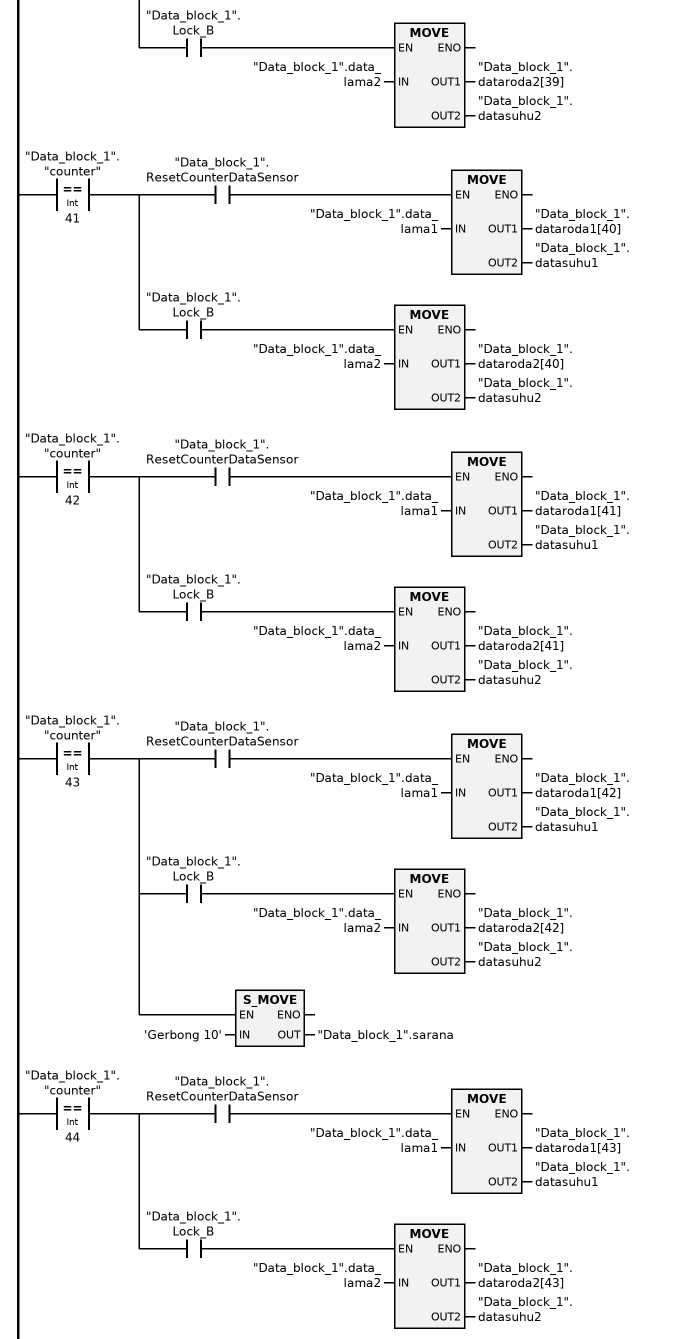
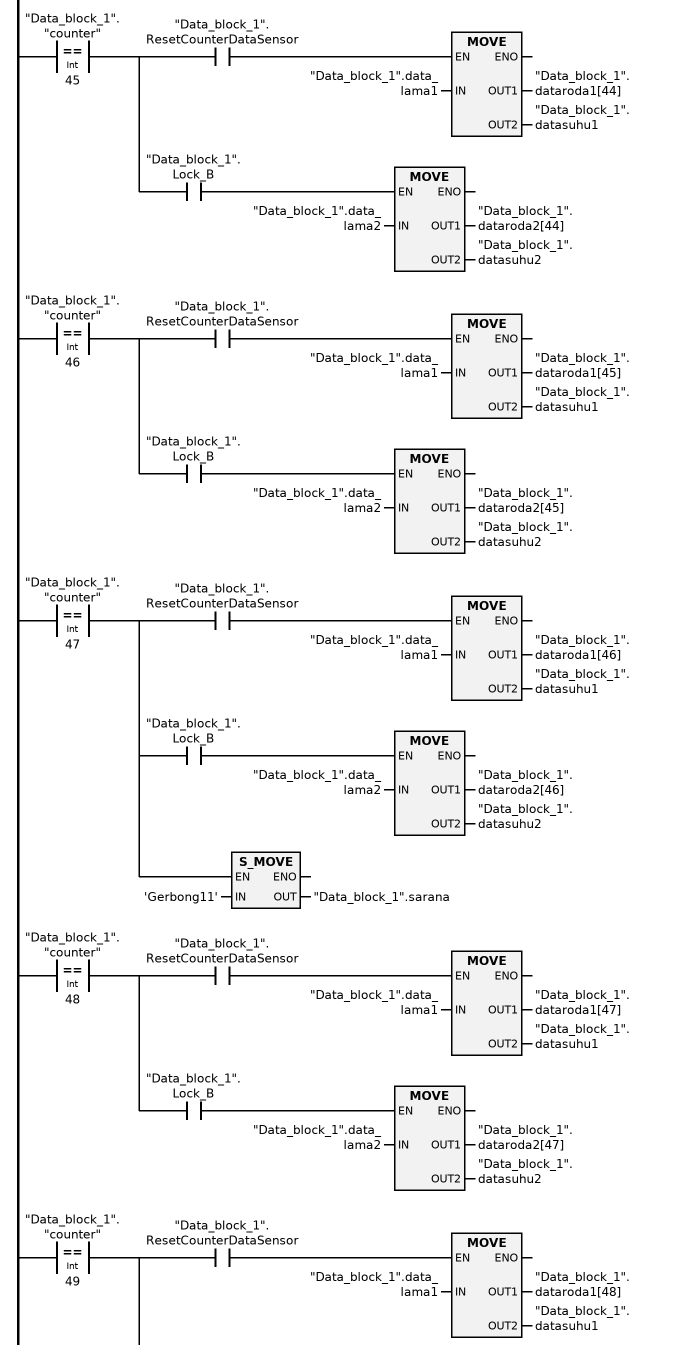
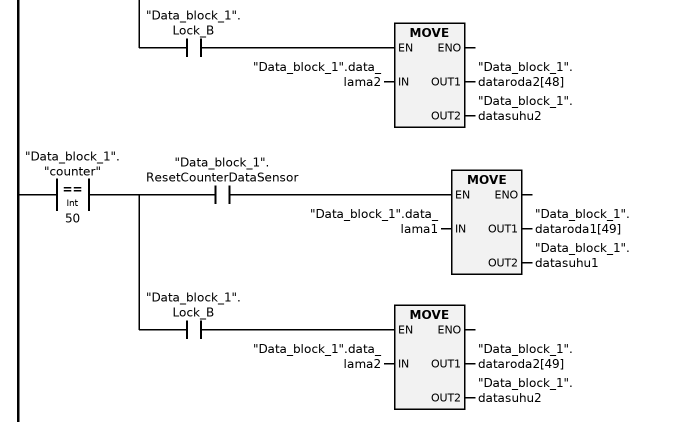
   #_w1 := "Data_block_1"."counter" = 1;
   IF #_w1 AND "Data_block_1".ResetCounterDataSensor THEN
       "Data_block_1".dataroda1[0] := "Data_block_1".data_lama1;
       "Data_block_1".datasuhu1 := "Data_block_1".data_lama1;
   END_IF;
   IF #_w1 AND "Data_block_1".Lock_B THEN
       "Data_block_1".dataroda2[0] := "Data_block_1".data_lama2;
       "Data_block_1".datasuhu2 := "Data_block_1".data_lama2;
   END_IF;
   IF #_w1 THEN S_MOVE(in := 'Lokomotif', out => "Data_block_1".sarana); END_IF;
   #_w2 := "Data_block_1"."counter" = 2;
   IF #_w2 AND "Data_block_1".ResetCounterDataSensor THEN
       "Data_block_1".dataroda1[1] := "Data_block_1".data_lama1;
       "Data_block_1".datasuhu1 := "Data_block_1".data_lama1;
   END_IF;
   IF #_w2 AND "Data_block_1".Lock_B THEN
       "Data_block_1".dataroda2[1] := "Data_block_1".data_lama2;
       "Data_block_1".datasuhu2 := "Data_block_1".data_lama2;
   END_IF;
   #_w3 := "Data_block_1"."counter" = 3;
   IF #_w3 AND "Data_block_1".ResetCounterDataSensor THEN
       "Data_block_1".dataroda1[2] := "Data_block_1".data_lama1;
       "Data_block_1".datasuhu1 := "Data_block_1".data_lama1;
   END_IF;
   IF #_w3 AND "Data_block_1".Lock_B THEN
       "Data_block_1".dataroda2[2] := "Data_block_1".data_lama2;
       "Data_block_1".datasuhu2 := "Data_block_1".data_lama2;
   END_IF;
   #_w4 := "Data_block_1"."counter" = 4;
   IF #_w4 AND "Data_block_1".ResetCounterDataSensor THEN
       "Data_block_1".dataroda1[3] := "Data_block_1".data_lama1;
       "Data_block_1".datasuhu1 := "Data_block_1".data_lama1;
   END_IF;
   IF #_w4 AND "Data_block_1".Lock_B THEN
       "Data_block_1".dataroda2[3] := "Data_block_1".data_lama2;
       "Data_block_1".datasuhu2 := "Data_block_1".data_lama2;
   END_IF;
   #_w5 := "Data_block_1"."counter" = 5;
   IF #_w5 AND "Data_block_1".ResetCounterDataSensor THEN
       "Data_block_1".dataroda1[4] := "Data_block_1".data_lama1;
       "Data_block_1".datasuhu1 := "Data_block_1".data_lama1;
   END_IF;
   IF #_w5 AND "Data_block_1".Lock_B THEN
       "Data_block_1".dataroda2[4] := "Data_block_1".data_lama2;
       "Data_block_1".datasuhu2 := "Data_block_1".data_lama2;
   END_IF;
   #_w6 := "Data_block_1"."counter" = 6;
   IF #_w6 AND "Data_block_1".ResetCounterDataSensor THEN
       "Data_block_1".dataroda1[5] := "Data_block_1".data_lama1;
       "Data_block_1".datasuhu1 := "Data_block_1".data_lama1;
   END_IF;
   IF #_w6 AND "Data_block_1".Lock_B THEN
       "Data_block_1".dataroda2[5] := "Data_block_1".data_lama2;
       "Data_block_1".datasuhu2 := "Data_block_1".data_lama2;
   END_IF;
   #_w7 := "Data_block_1"."counter" = 7;
   IF #_w7 AND "Data_block_1".ResetCounterDataSensor THEN
       "Data_block_1".dataroda1[6] := "Data_block_1".data_lama1;
       "Data_block_1".datasuhu1 := "Data_block_1".data_lama1;
   END_IF;
   IF #_w7 AND "Data_block_1".Lock_B THEN
       "Data_block_1".dataroda2[6] := "Data_block_1".data_lama2;
       "Data_block_1".datasuhu2 := "Data_block_1".data_lama2;
   END_IF;
   IF #_w7 THEN S_MOVE(in := 'Gerbong 1', out => "Data_block_1".sarana); END_IF;
   #_w8 := "Data_block_1"."counter" = 8;
   IF #_w8 AND "Data_block_1".ResetCounterDataSensor THEN
       "Data_block_1".dataroda1[7] := "Data_block_1".data_lama1;
       "Data_block_1".datasuhu1 := "Data_block_1".data_lama1;
   END_IF;
   IF #_w8 AND "Data_block_1".Lock_B THEN
       "Data_block_1".dataroda2[7] := "Data_block_1".data_lama2;
       "Data_block_1".datasuhu2 := "Data_block_1".data_lama2;
   END_IF;
   #_w9 := "Data_block_1"."counter" = 9;
   IF #_w9 AND "Data_block_1".ResetCounterDataSensor THEN
       "Data_block_1".dataroda1[8] := "Data_block_1".data_lama1;
       "Data_block_1".datasuhu1 := "Data_block_1".data_lama1;
   END_IF;
   IF #_w9 AND "Data_block_1".Lock_B THEN
       "Data_block_1".dataroda2[8] := "Data_block_1".data_lama2;
       "Data_block_1".datasuhu2 := "Data_block_1".data_lama2;
   END_IF;
   #_w10 := "Data_block_1"."counter" = 10;
   IF #_w10 AND "Data_block_1".ResetCounterDataSensor THEN
       "Data_block_1".dataroda1[9] := "Data_block_1".data_lama1;
       "Data_block_1".datasuhu1 := "Data_block_1".data_lama1;
   END_IF;
   IF #_w10 AND "Data_block_1".Lock_B THEN
       "Data_block_1".dataroda2[9] := "Data_block_1".data_lama2;
       "Data_block_1".datasuhu2 := "Data_block_1".data_lama2;
   END_IF;
   #_w11 := "Data_block_1"."counter" = 11;
   IF #_w11 AND "Data_block_1".ResetCounterDataSensor THEN
       "Data_block_1".dataroda1[10] := "Data_block_1".data_lama1;
       "Data_block_1".datasuhu1 := "Data_block_1".data_lama1;
   END_IF;
   IF #_w11 AND "Data_block_1".Lock_B THEN
       "Data_block_1".dataroda2[10] := "Data_block_1".data_lama2;
       "Data_block_1".datasuhu2 := "Data_block_1".data_lama2;
   END_IF;
   IF #_w11 THEN S_MOVE(in := 'Gerbong 2', out => "Data_block_1".sarana); END_IF;
   #_w12 := "Data_block_1"."counter" = 12;
   IF #_w12 AND "Data_block_1".ResetCounterDataSensor THEN
       "Data_block_1".dataroda1[11] := "Data_block_1".data_lama1;
       "Data_block_1".datasuhu1 := "Data_block_1".data_lama1;
   END_IF;
   IF #_w12 AND "Data_block_1".Lock_B THEN
       "Data_block_1".dataroda2[11] := "Data_block_1".data_lama2;
       "Data_block_1".datasuhu2 := "Data_block_1".data_lama2;
   END_IF;
   #_w13 := "Data_block_1"."counter" = 13;
   IF #_w13 AND "Data_block_1".ResetCounterDataSensor THEN
       "Data_block_1".dataroda1[12] := "Data_block_1".data_lama1;
       "Data_block_1".datasuhu1 := "Data_block_1".data_lama1;
   END_IF;
   IF #_w13 AND "Data_block_1".Lock_B THEN
       "Data_block_1".dataroda2[12] := "Data_block_1".data_lama2;
       "Data_block_1".datasuhu2 := "Data_block_1".data_lama2;
   END_IF;
   #_w14 := "Data_block_1"."counter" = 14;
   IF #_w14 AND "Data_block_1".ResetCounterDataSensor THEN
       "Data_block_1".dataroda1[13] := "Data_block_1".data_lama1;
       "Data_block_1".datasuhu1 := "Data_block_1".data_lama1;
   END_IF;
   IF #_w14 AND "Data_block_1".Lock_B THEN
       "Data_block_1".dataroda2[13] := "Data_block_1".data_lama2;
       "Data_block_1".datasuhu2 := "Data_block_1".data_lama2;
   END_IF;
   #_w15 := "Data_block_1"."counter" = 15;
   IF #_w15 AND "Data_block_1".ResetCounterDataSensor THEN
       "Data_block_1".dataroda1[14] := "Data_block_1".data_lama1;
       "Data_block_1".datasuhu1 := "Data_block_1".data_lama1;
   END_IF;
   IF #_w15 AND "Data_block_1".Lock_B THEN
       "Data_block_1".dataroda2[14] := "Data_block_1".data_lama2;
       "Data_block_1".datasuhu2 := "Data_block_1".data_lama2;
   END_IF;
   IF #_w15 THEN S_MOVE(in := 'Gerbong 3', out => "Data_block_1".sarana); END_IF;
   #_w16 := "Data_block_1"."counter" = 16;
   IF #_w16 AND "Data_block_1".ResetCounterDataSensor THEN
       "Data_block_1".dataroda1[15] := "Data_block_1".data_lama1;
       "Data_block_1".datasuhu1 := "Data_block_1".data_lama1;
   END_IF;
   IF #_w16 AND "Data_block_1".Lock_B THEN
       "Data_block_1".dataroda2[15] := "Data_block_1".data_lama2;
       "Data_block_1".datasuhu2 := "Data_block_1".data_lama2;
   END_IF;
   #_w17 := "Data_block_1"."counter" = 17;
   IF #_w17 AND "Data_block_1".ResetCounterDataSensor THEN
       "Data_block_1".dataroda1[16] := "Data_block_1".data_lama1;
       "Data_block_1".datasuhu1 := "Data_block_1".data_lama1;
   END_IF;
   IF #_w17 AND "Data_block_1".Lock_B THEN
       "Data_block_1".dataroda2[16] := "Data_block_1".data_lama2;
       "Data_block_1".datasuhu2 := "Data_block_1".data_lama2;
   END_IF;
   #_w18 := "Data_block_1"."counter" = 18;
   IF #_w18 AND "Data_block_1".ResetCounterDataSensor THEN
       "Data_block_1".dataroda1[17] := "Data_block_1".data_lama1;
       "Data_block_1".datasuhu1 := "Data_block_1".data_lama1;
   END_IF;
   IF #_w18 AND "Data_block_1".Lock_B THEN
       "Data_block_1".dataroda2[17] := "Data_block_1".data_lama2;
       "Data_block_1".datasuhu2 := "Data_block_1".data_lama2;
   END_IF;
   #_w19 := "Data_block_1"."counter" = 19;
   IF #_w19 AND "Data_block_1".ResetCounterDataSensor THEN
       "Data_block_1".dataroda1[18] := "Data_block_1".data_lama1;
       "Data_block_1".datasuhu1 := "Data_block_1".data_lama1;
   END_IF;
   IF #_w19 AND "Data_block_1".Lock_B THEN
       "Data_block_1".dataroda2[18] := "Data_block_1".data_lama2;
       "Data_block_1".datasuhu2 := "Data_block_1".data_lama2;
   END_IF;
   IF #_w19 THEN S_MOVE(in := 'Gerbong 4', out => "Data_block_1".sarana); END_IF;
   #_w20 := "Data_block_1"."counter" = 20;
   IF #_w20 AND "Data_block_1".ResetCounterDataSensor THEN
       "Data_block_1".dataroda1[19] := "Data_block_1".data_lama1;
       "Data_block_1".datasuhu1 := "Data_block_1".data_lama1;
   END_IF;
   IF #_w20 AND "Data_block_1".Lock_B THEN
       "Data_block_1".dataroda2[19] := "Data_block_1".data_lama2;
       "Data_block_1".datasuhu2 := "Data_block_1".data_lama2;
   END_IF;
   #_w21 := "Data_block_1"."counter" = 21;
   IF #_w21 AND "Data_block_1".ResetCounterDataSensor THEN
       "Data_block_1".dataroda1[20] := "Data_block_1".data_lama1;
       "Data_block_1".datasuhu1 := "Data_block_1".data_lama1;
   END_IF;
   IF #_w21 AND "Data_block_1".Lock_B THEN
       "Data_block_1".dataroda2[20] := "Data_block_1".data_lama2;
       "Data_block_1".datasuhu2 := "Data_block_1".data_lama2;
   END_IF;
   #_w22 := "Data_block_1"."counter" = 22;
   IF #_w22 AND "Data_block_1".ResetCounterDataSensor THEN
       "Data_block_1".dataroda1[21] := "Data_block_1".data_lama1;
       "Data_block_1".datasuhu1 := "Data_block_1".data_lama1;
   END_IF;
   IF #_w22 AND "Data_block_1".Lock_B THEN
       "Data_block_1".dataroda2[21] := "Data_block_1".data_lama2;
       "Data_block_1".datasuhu2 := "Data_block_1".data_lama2;
   END_IF;
   #_w23 := "Data_block_1"."counter" = 23;
   IF #_w23 AND "Data_block_1".ResetCounterDataSensor THEN
       "Data_block_1".dataroda1[22] := "Data_block_1".data_lama1;
       "Data_block_1".datasuhu1 := "Data_block_1".data_lama1;
   END_IF;
   IF #_w23 AND "Data_block_1".Lock_B THEN
       "Data_block_1".dataroda2[22] := "Data_block_1".data_lama2;
       "Data_block_1".datasuhu2 := "Data_block_1".data_lama2;
   END_IF;
   IF #_w23 THEN S_MOVE(in := 'Gerbong 5', out => "Data_block_1".sarana); END_IF;
   #_w24 := "Data_block_1"."counter" = 24;
   IF #_w24 AND "Data_block_1".ResetCounterDataSensor THEN
       "Data_block_1".dataroda1[23] := "Data_block_1".data_lama1;
       "Data_block_1".datasuhu1 := "Data_block_1".data_lama1;
   END_IF;
   IF #_w24 AND "Data_block_1".Lock_B THEN
       "Data_block_1".dataroda2[23] := "Data_block_1".data_lama2;
       "Data_block_1".datasuhu2 := "Data_block_1".data_lama2;
   END_IF;
   #_w25 := "Data_block_1"."counter" = 25;
   IF #_w25 AND "Data_block_1".ResetCounterDataSensor THEN
       "Data_block_1".dataroda1[24] := "Data_block_1".data_lama1;
       "Data_block_1".datasuhu1 := "Data_block_1".data_lama1;
   END_IF;
   IF #_w25 AND "Data_block_1".Lock_B THEN
       "Data_block_1".dataroda2[24] := "Data_block_1".data_lama2;
       "Data_block_1".datasuhu2 := "Data_block_1".data_lama2;
   END_IF;
   #_w26 := "Data_block_1"."counter" = 26;
   IF #_w26 AND "Data_block_1".ResetCounterDataSensor THEN
       "Data_block_1".dataroda1[25] := "Data_block_1".data_lama1;
       "Data_block_1".datasuhu1 := "Data_block_1".data_lama1;
   END_IF;
   IF #_w26 AND "Data_block_1".Lock_B THEN
       "Data_block_1".dataroda2[25] := "Data_block_1".data_lama2;
       "Data_block_1".datasuhu2 := "Data_block_1".data_lama2;
   END_IF;
   #_w27 := "Data_block_1"."counter" = 27;
   IF #_w27 AND "Data_block_1".ResetCounterDataSensor THEN
       "Data_block_1".dataroda1[26] := "Data_block_1".data_lama1;
       "Data_block_1".datasuhu1 := "Data_block_1".data_lama1;
   END_IF;
   IF #_w27 AND "Data_block_1".Lock_B THEN
       "Data_block_1".dataroda2[26] := "Data_block_1".data_lama2;
       "Data_block_1".datasuhu2 := "Data_block_1".data_lama2;
   END_IF;
   IF #_w27 THEN S_MOVE(in := 'Gerbong 6', out => "Data_block_1".sarana); END_IF;
   #_w28 := "Data_block_1"."counter" = 28;
   IF #_w28 AND "Data_block_1".ResetCounterDataSensor THEN
       "Data_block_1".dataroda1[27] := "Data_block_1".data_lama1;
       "Data_block_1".datasuhu1 := "Data_block_1".data_lama1;
   END_IF;
   IF #_w28 AND "Data_block_1".Lock_B THEN
       "Data_block_1".dataroda2[27] := "Data_block_1".data_lama2;
       "Data_block_1".datasuhu2 := "Data_block_1".data_lama2;
   END_IF;
   #_w29 := "Data_block_1"."counter" = 29;
   IF #_w29 AND "Data_block_1".ResetCounterDataSensor THEN
       "Data_block_1".dataroda1[28] := "Data_block_1".data_lama1;
       "Data_block_1".datasuhu1 := "Data_block_1".data_lama1;
   END_IF;
   IF #_w29 AND "Data_block_1".Lock_B THEN
       "Data_block_1".dataroda2[28] := "Data_block_1".data_lama2;
       "Data_block_1".datasuhu2 := "Data_block_1".data_lama2;
   END_IF;
   #_w30 := "Data_block_1"."counter" = 30;
   IF #_w30 AND "Data_block_1".ResetCounterDataSensor THEN
       "Data_block_1".dataroda1[29] := "Data_block_1".data_lama1;
       "Data_block_1".datasuhu1 := "Data_block_1".data_lama1;
   END_IF;
   IF #_w30 AND "Data_block_1".Lock_B THEN
       "Data_block_1".dataroda2[29] := "Data_block_1".data_lama2;
       "Data_block_1".datasuhu2 := "Data_block_1".data_lama2;
   END_IF;
   #_w31 := "Data_block_1"."counter" = 31;
   IF #_w31 AND "Data_block_1".ResetCounterDataSensor THEN
       "Data_block_1".dataroda1[30] := "Data_block_1".data_lama1;
       "Data_block_1".datasuhu1 := "Data_block_1".data_lama1;
   END_IF;
   IF #_w31 AND "Data_block_1".Lock_B THEN
       "Data_block_1".dataroda2[30] := "Data_block_1".data_lama2;
       "Data_block_1".datasuhu2 := "Data_block_1".data_lama2;
   END_IF;
   IF #_w31 THEN S_MOVE(in := 'Gerbong 7', out => "Data_block_1".sarana); END_IF;
   #_w32 := "Data_block_1"."counter" = 32;
   IF #_w32 AND "Data_block_1".ResetCounterDataSensor THEN
       "Data_block_1".dataroda1[31] := "Data_block_1".data_lama1;
       "Data_block_1".datasuhu1 := "Data_block_1".data_lama1;
   END_IF;
   IF #_w32 AND "Data_block_1".Lock_B THEN
       "Data_block_1".dataroda2[31] := "Data_block_1".data_lama2;
       "Data_block_1".datasuhu2 := "Data_block_1".data_lama2;
   END_IF;
   #_w33 := "Data_block_1"."counter" = 33;
   IF #_w33 AND "Data_block_1".ResetCounterDataSensor THEN
       "Data_block_1".dataroda1[32] := "Data_block_1".data_lama1;
       "Data_block_1".datasuhu1 := "Data_block_1".data_lama1;
   END_IF;
   IF #_w33 AND "Data_block_1".Lock_B THEN
       "Data_block_1".dataroda2[32] := "Data_block_1".data_lama2;
       "Data_block_1".datasuhu2 := "Data_block_1".data_lama2;
   END_IF;
   #_w34 := "Data_block_1"."counter" = 34;
   IF #_w34 AND "Data_block_1".ResetCounterDataSensor THEN
       "Data_block_1".dataroda1[33] := "Data_block_1".data_lama1;
       "Data_block_1".datasuhu1 := "Data_block_1".data_lama1;
   END_IF;
   IF #_w34 AND "Data_block_1".Lock_B THEN
       "Data_block_1".dataroda2[33] := "Data_block_1".data_lama2;
       "Data_block_1".datasuhu2 := "Data_block_1".data_lama2;
   END_IF;
   #_w35 := "Data_block_1"."counter" = 35;
   IF #_w35 AND "Data_block_1".ResetCounterDataSensor THEN
       "Data_block_1".dataroda1[34] := "Data_block_1".data_lama1;
       "Data_block_1".datasuhu1 := "Data_block_1".data_lama1;
   END_IF;
   IF #_w35 AND "Data_block_1".Lock_B THEN
       "Data_block_1".dataroda2[34] := "Data_block_1".data_lama2;
       "Data_block_1".datasuhu2 := "Data_block_1".data_lama2;
   END_IF;
   IF #_w35 THEN S_MOVE(in := 'Gerbong 8', out => "Data_block_1".sarana); END_IF;
   #_w36 := "Data_block_1"."counter" = 36;
   IF #_w36 AND "Data_block_1".ResetCounterDataSensor THEN
       "Data_block_1".dataroda1[35] := "Data_block_1".data_lama1;
       "Data_block_1".datasuhu1 := "Data_block_1".data_lama1;
   END_IF;
   IF #_w36 AND "Data_block_1".Lock_B THEN
       "Data_block_1".dataroda2[35] := "Data_block_1".data_lama2;
       "Data_block_1".datasuhu2 := "Data_block_1".data_lama2;
   END_IF;
   #_w37 := "Data_block_1"."counter" = 37;
   IF #_w37 AND "Data_block_1".ResetCounterDataSensor THEN
       "Data_block_1".dataroda1[36] := "Data_block_1".data_lama1;
       "Data_block_1".datasuhu1 := "Data_block_1".data_lama1;
   END_IF;
   IF #_w37 AND "Data_block_1".Lock_B THEN
       "Data_block_1".dataroda2[36] := "Data_block_1".data_lama2;
       "Data_block_1".datasuhu2 := "Data_block_1".data_lama2;
   END_IF;
   #_w38 := "Data_block_1"."counter" = 38;
   IF #_w38 AND "Data_block_1".ResetCounterDataSensor THEN
       "Data_block_1".dataroda1[37] := "Data_block_1".data_lama1;
       "Data_block_1".datasuhu1 := "Data_block_1".data_lama1;
   END_IF;
   IF #_w38 AND "Data_block_1".Lock_B THEN
       "Data_block_1".dataroda2[37] := "Data_block_1".data_lama2;
       "Data_block_1".datasuhu2 := "Data_block_1".data_lama2;
   END_IF;
   #_w39 := "Data_block_1"."counter" = 39;
   IF #_w39 AND "Data_block_1".ResetCounterDataSensor THEN
       "Data_block_1".dataroda1[38] := "Data_block_1".data_lama1;
       "Data_block_1".datasuhu1 := "Data_block_1".data_lama1;
   END_IF;
   IF #_w39 AND "Data_block_1".Lock_B THEN
       "Data_block_1".dataroda2[38] := "Data_block_1".data_lama2;
       "Data_block_1".datasuhu2 := "Data_block_1".data_lama2;
   END_IF;
   IF #_w39 THEN S_MOVE(in := 'Gerbong 9', out => "Data_block_1".sarana); END_IF;
   #_w40 := "Data_block_1"."counter" = 40;
   IF #_w40 AND "Data_block_1".ResetCounterDataSensor THEN
       "Data_block_1".dataroda1[39] := "Data_block_1".data_lama1;
       "Data_block_1".datasuhu1 := "Data_block_1".data_lama1;
   END_IF;
   IF #_w40 AND "Data_block_1".Lock_B THEN
       "Data_block_1".dataroda2[39] := "Data_block_1".data_lama2;
       "Data_block_1".datasuhu2 := "Data_block_1".data_lama2;
   END_IF;
   #_w41 := "Data_block_1"."counter" = 41;
   IF #_w41 AND "Data_block_1".ResetCounterDataSensor THEN
       "Data_block_1".dataroda1[40] := "Data_block_1".data_lama1;
       "Data_block_1".datasuhu1 := "Data_block_1".data_lama1;
   END_IF;
   IF #_w41 AND "Data_block_1".Lock_B THEN
       "Data_block_1".dataroda2[40] := "Data_block_1".data_lama2;
       "Data_block_1".datasuhu2 := "Data_block_1".data_lama2;
   END_IF;
   #_w42 := "Data_block_1"."counter" = 42;
   IF #_w42 AND "Data_block_1".ResetCounterDataSensor THEN
       "Data_block_1".dataroda1[41] := "Data_block_1".data_lama1;
       "Data_block_1".datasuhu1 := "Data_block_1".data_lama1;
   END_IF;
   IF #_w42 AND "Data_block_1".Lock_B THEN
       "Data_block_1".dataroda2[41] := "Data_block_1".data_lama2;
       "Data_block_1".datasuhu2 := "Data_block_1".data_lama2;
   END_IF;
   #_w43 := "Data_block_1"."counter" = 43;
   IF #_w43 AND "Data_block_1".ResetCounterDataSensor THEN
       "Data_block_1".dataroda1[42] := "Data_block_1".data_lama1;
       "Data_block_1".datasuhu1 := "Data_block_1".data_lama1;
   END_IF;
   IF #_w43 AND "Data_block_1".Lock_B THEN
       "Data_block_1".dataroda2[42] := "Data_block_1".data_lama2;
       "Data_block_1".datasuhu2 := "Data_block_1".data_lama2;
   END_IF;
   IF #_w43 THEN S_MOVE(in := 'Gerbong 10', out => "Data_block_1".sarana); END_IF;
   #_w44 := "Data_block_1"."counter" = 44;
   IF #_w44 AND "Data_block_1".ResetCounterDataSensor THEN
       "Data_block_1".dataroda1[43] := "Data_block_1".data_lama1;
       "Data_block_1".datasuhu1 := "Data_block_1".data_lama1;
   END_IF;
   IF #_w44 AND "Data_block_1".Lock_B THEN
       "Data_block_1".dataroda2[43] := "Data_block_1".data_lama2;
       "Data_block_1".datasuhu2 := "Data_block_1".data_lama2;
   END_IF;
   #_w45 := "Data_block_1"."counter" = 45;
   IF #_w45 AND "Data_block_1".ResetCounterDataSensor THEN
       "Data_block_1".dataroda1[44] := "Data_block_1".data_lama1;
       "Data_block_1".datasuhu1 := "Data_block_1".data_lama1;
   END_IF;
   IF #_w45 AND "Data_block_1".Lock_B THEN
       "Data_block_1".dataroda2[44] := "Data_block_1".data_lama2;
       "Data_block_1".datasuhu2 := "Data_block_1".data_lama2;
   END_IF;
   #_w46 := "Data_block_1"."counter" = 46;
   IF #_w46 AND "Data_block_1".ResetCounterDataSensor THEN
       "Data_block_1".dataroda1[45] := "Data_block_1".data_lama1;
       "Data_block_1".datasuhu1 := "Data_block_1".data_lama1;
   END_IF;
   IF #_w46 AND "Data_block_1".Lock_B THEN
       "Data_block_1".dataroda2[45] := "Data_block_1".data_lama2;
       "Data_block_1".datasuhu2 := "Data_block_1".data_lama2;
   END_IF;
   #_w47 := "Data_block_1"."counter" = 47;
   IF #_w47 AND "Data_block_1".ResetCounterDataSensor THEN
       "Data_block_1".dataroda1[46] := "Data_block_1".data_lama1;
       "Data_block_1".datasuhu1 := "Data_block_1".data_lama1;
   END_IF;
   IF #_w47 AND "Data_block_1".Lock_B THEN
       "Data_block_1".dataroda2[46] := "Data_block_1".data_lama2;
       "Data_block_1".datasuhu2 := "Data_block_1".data_lama2;
   END_IF;
   IF #_w47 THEN S_MOVE(in := 'Gerbong11', out => "Data_block_1".sarana); END_IF;
   #_w48 := "Data_block_1"."counter" = 48;
   IF #_w48 AND "Data_block_1".ResetCounterDataSensor THEN
       "Data_block_1".dataroda1[47] := "Data_block_1".data_lama1;
       "Data_block_1".datasuhu1 := "Data_block_1".data_lama1;
   END_IF;
   IF #_w48 AND "Data_block_1".Lock_B THEN
       "Data_block_1".dataroda2[47] := "Data_block_1".data_lama2;
       "Data_block_1".datasuhu2 := "Data_block_1".data_lama2;
   END_IF;
   #_w49 := "Data_block_1"."counter" = 49;
   IF #_w49 AND "Data_block_1".ResetCounterDataSensor THEN
       "Data_block_1".dataroda1[48] := "Data_block_1".data_lama1;
       "Data_block_1".datasuhu1 := "Data_block_1".data_lama1;
   END_IF;
   IF #_w49 AND "Data_block_1".Lock_B THEN
       "Data_block_1".dataroda2[48] := "Data_block_1".data_lama2;
       "Data_block_1".datasuhu2 := "Data_block_1".data_lama2;
   END_IF;
   #_w50 := "Data_block_1"."counter" = 50;
   IF #_w50 AND "Data_block_1".ResetCounterDataSensor THEN
       "Data_block_1".dataroda1[49] := "Data_block_1".data_lama1;
       "Data_block_1".datasuhu1 := "Data_block_1".data_lama1;
   END_IF;
   IF #_w50 AND "Data_block_1".Lock_B THEN
       "Data_block_1".dataroda2[49] := "Data_block_1".data_lama2;
       "Data_block_1".datasuhu2 := "Data_block_1".data_lama2;
   END_IF;
END_REGION

REGION Network 13: reset data suhu roda
   // ketika reset aktif 
   // 
   // - maka datasuhu, array data suhu roda akan kembali 0
   // - maka counter genap kembali 0
   // - maka counter ganjil menjadi -1
   // - maka sarana akan kosong
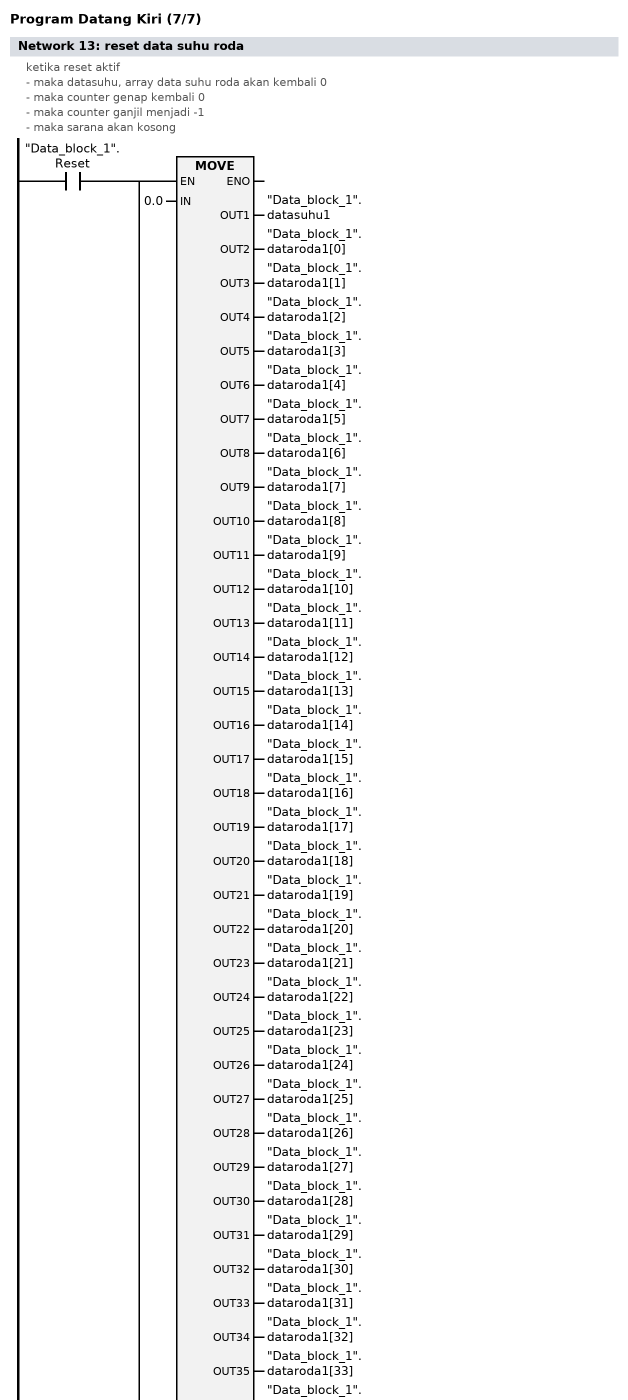
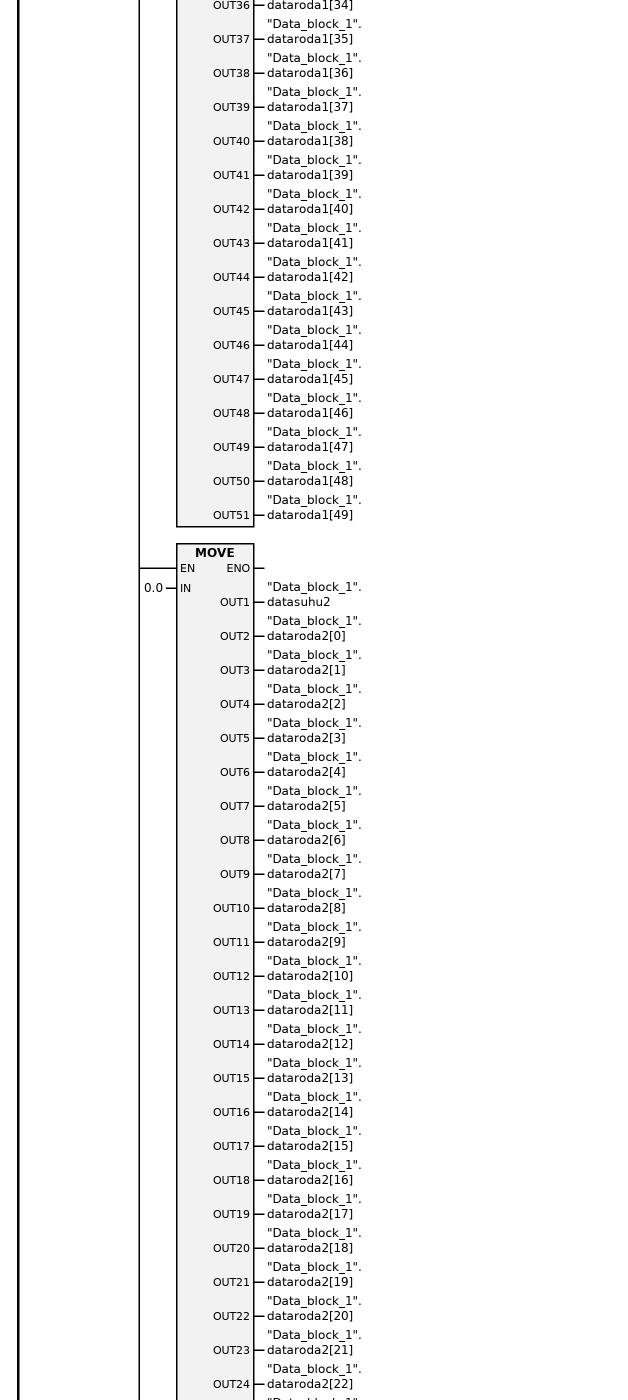
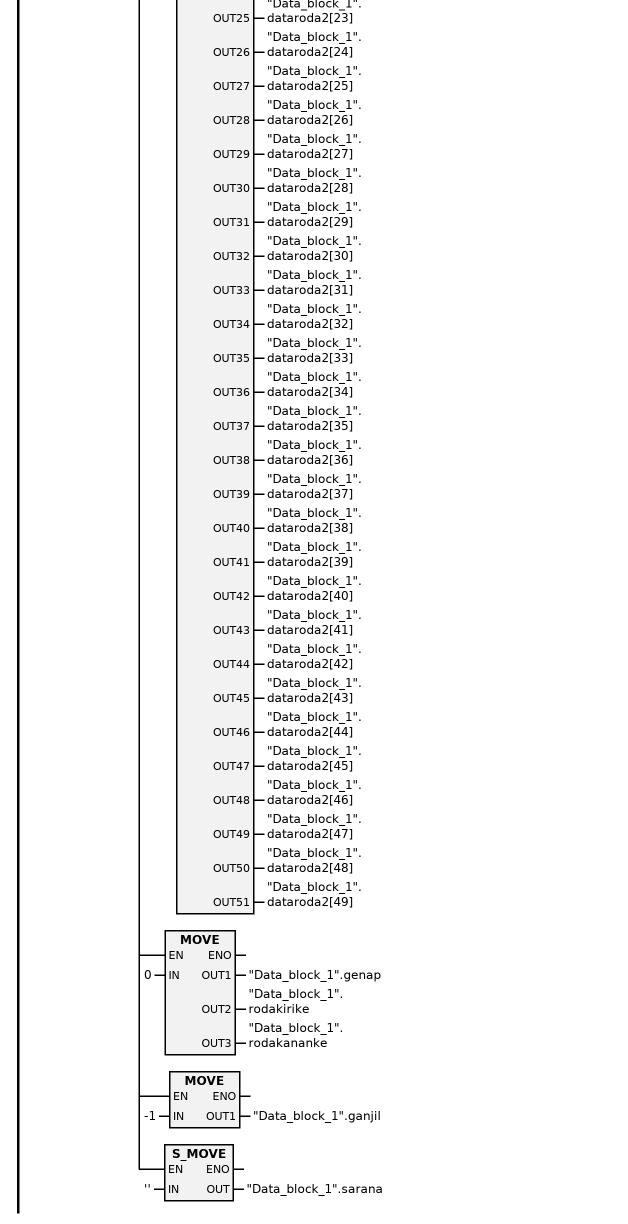
   IF "Data_block_1".Reset THEN
       "Data_block_1".datasuhu1 := 0.0;
       "Data_block_1".dataroda1[0] := 0.0;
       "Data_block_1".dataroda1[1] := 0.0;
       "Data_block_1".dataroda1[2] := 0.0;
       "Data_block_1".dataroda1[3] := 0.0;
       "Data_block_1".dataroda1[4] := 0.0;
       "Data_block_1".dataroda1[5] := 0.0;
       "Data_block_1".dataroda1[6] := 0.0;
       "Data_block_1".dataroda1[7] := 0.0;
       "Data_block_1".dataroda1[8] := 0.0;
       "Data_block_1".dataroda1[9] := 0.0;
       "Data_block_1".dataroda1[10] := 0.0;
       "Data_block_1".dataroda1[11] := 0.0;
       "Data_block_1".dataroda1[12] := 0.0;
       "Data_block_1".dataroda1[13] := 0.0;
       "Data_block_1".dataroda1[14] := 0.0;
       "Data_block_1".dataroda1[15] := 0.0;
       "Data_block_1".dataroda1[16] := 0.0;
       "Data_block_1".dataroda1[17] := 0.0;
       "Data_block_1".dataroda1[18] := 0.0;
       "Data_block_1".dataroda1[19] := 0.0;
       "Data_block_1".dataroda1[20] := 0.0;
       "Data_block_1".dataroda1[21] := 0.0;
       "Data_block_1".dataroda1[22] := 0.0;
       "Data_block_1".dataroda1[23] := 0.0;
       "Data_block_1".dataroda1[24] := 0.0;
       "Data_block_1".dataroda1[25] := 0.0;
       "Data_block_1".dataroda1[26] := 0.0;
       "Data_block_1".dataroda1[27] := 0.0;
       "Data_block_1".dataroda1[28] := 0.0;
       "Data_block_1".dataroda1[29] := 0.0;
       "Data_block_1".dataroda1[30] := 0.0;
       "Data_block_1".dataroda1[31] := 0.0;
       "Data_block_1".dataroda1[32] := 0.0;
       "Data_block_1".dataroda1[33] := 0.0;
       "Data_block_1".dataroda1[34] := 0.0;
       "Data_block_1".dataroda1[35] := 0.0;
       "Data_block_1".dataroda1[36] := 0.0;
       "Data_block_1".dataroda1[37] := 0.0;
       "Data_block_1".dataroda1[38] := 0.0;
       "Data_block_1".dataroda1[39] := 0.0;
       "Data_block_1".dataroda1[40] := 0.0;
       "Data_block_1".dataroda1[41] := 0.0;
       "Data_block_1".dataroda1[42] := 0.0;
       "Data_block_1".dataroda1[43] := 0.0;
       "Data_block_1".dataroda1[44] := 0.0;
       "Data_block_1".dataroda1[45] := 0.0;
       "Data_block_1".dataroda1[46] := 0.0;
       "Data_block_1".dataroda1[47] := 0.0;
       "Data_block_1".dataroda1[48] := 0.0;
       "Data_block_1".dataroda1[49] := 0.0;
       "Data_block_1".datasuhu2 := 0.0;
       "Data_block_1".dataroda2[0] := 0.0;
       "Data_block_1".dataroda2[1] := 0.0;
       "Data_block_1".dataroda2[2] := 0.0;
       "Data_block_1".dataroda2[3] := 0.0;
       "Data_block_1".dataroda2[4] := 0.0;
       "Data_block_1".dataroda2[5] := 0.0;
       "Data_block_1".dataroda2[6] := 0.0;
       "Data_block_1".dataroda2[7] := 0.0;
       "Data_block_1".dataroda2[8] := 0.0;
       "Data_block_1".dataroda2[9] := 0.0;
       "Data_block_1".dataroda2[10] := 0.0;
       "Data_block_1".dataroda2[11] := 0.0;
       "Data_block_1".dataroda2[12] := 0.0;
       "Data_block_1".dataroda2[13] := 0.0;
       "Data_block_1".dataroda2[14] := 0.0;
       "Data_block_1".dataroda2[15] := 0.0;
       "Data_block_1".dataroda2[16] := 0.0;
       "Data_block_1".dataroda2[17] := 0.0;
       "Data_block_1".dataroda2[18] := 0.0;
       "Data_block_1".dataroda2[19] := 0.0;
       "Data_block_1".dataroda2[20] := 0.0;
       "Data_block_1".dataroda2[21] := 0.0;
       "Data_block_1".dataroda2[22] := 0.0;
       "Data_block_1".dataroda2[23] := 0.0;
       "Data_block_1".dataroda2[24] := 0.0;
       "Data_block_1".dataroda2[25] := 0.0;
       "Data_block_1".dataroda2[26] := 0.0;
       "Data_block_1".dataroda2[27] := 0.0;
       "Data_block_1".dataroda2[28] := 0.0;
       "Data_block_1".dataroda2[29] := 0.0;
       "Data_block_1".dataroda2[30] := 0.0;
       "Data_block_1".dataroda2[31] := 0.0;
       "Data_block_1".dataroda2[32] := 0.0;
       "Data_block_1".dataroda2[33] := 0.0;
       "Data_block_1".dataroda2[34] := 0.0;
       "Data_block_1".dataroda2[35] := 0.0;
       "Data_block_1".dataroda2[36] := 0.0;
       "Data_block_1".dataroda2[37] := 0.0;
       "Data_block_1".dataroda2[38] := 0.0;
       "Data_block_1".dataroda2[39] := 0.0;
       "Data_block_1".dataroda2[40] := 0.0;
       "Data_block_1".dataroda2[41] := 0.0;
       "Data_block_1".dataroda2[42] := 0.0;
       "Data_block_1".dataroda2[43] := 0.0;
       "Data_block_1".dataroda2[44] := 0.0;
       "Data_block_1".dataroda2[45] := 0.0;
       "Data_block_1".dataroda2[46] := 0.0;
       "Data_block_1".dataroda2[47] := 0.0;
       "Data_block_1".dataroda2[48] := 0.0;
       "Data_block_1".dataroda2[49] := 0.0;
       "Data_block_1".genap := 0;
       "Data_block_1".rodakirike := 0;
       "Data_block_1".rodakananke := 0;
       "Data_block_1".ganjil := -1;
       S_MOVE(in := '', out => "Data_block_1".sarana);
   END_IF;
END_REGION
END_ORGANIZATION_BLOCK

ORGANIZATION_BLOCK "Program Datang Kanan"   // OB123, LAD, ProgramCycle
TITLE = Datang Kanan
{ S7_Optimized_Access := 'TRUE' }
VERSION : 0.1
   VAR_INPUT
      Initial_Call : Bool;   // Initial call of this OB
      Remanence : Bool;   // =True, if remanent data are available
   END_VAR
   VAR_TEMP   // added for the SCL form of the ladder/FBD networks
      _w1 : Bool;
   END_VAR
BEGIN

REGION Network 1: Lock A
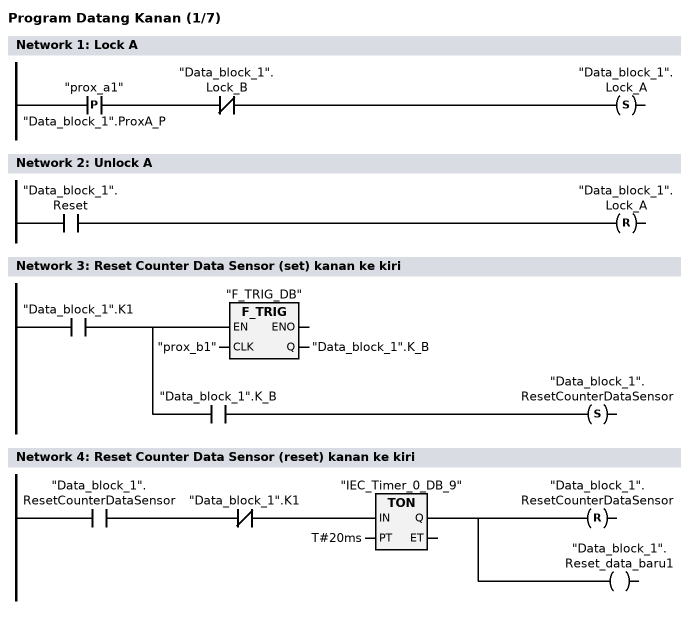
   RUNG wire#powerrail
      P_Contact(operand := "prox_a1", bit := "Data_block_1".ProxA_P)
      I_Contact( "Data_block_1".Lock_B )
      S_Coil( "Data_block_1".Lock_A )
   END_RUNG
   // the same network as SCL:
   #_w1 := "prox_a1" AND NOT "Data_block_1".ProxA_P;   // rising edge of "prox_a1"
   "Data_block_1".ProxA_P := "prox_a1";
   IF #_w1 AND NOT "Data_block_1".Lock_B THEN "Data_block_1".Lock_A := TRUE; END_IF;
END_REGION

REGION Network 2: Unlock A
   RUNG wire#powerrail
      Contact( "Data_block_1".Reset )
      R_Coil( "Data_block_1".Lock_A )
   END_RUNG
   // the same network as SCL:
   IF "Data_block_1".Reset THEN "Data_block_1".Lock_A := FALSE; END_IF;
END_REGION

REGION Network 3: Reset Counter Data Sensor (set) kanan ke kiri
   IF "Data_block_1".K1 THEN
       "F_TRIG_DB"(CLK := "prox_b1", Q => "Data_block_1".K_B);   // F_TRIG
   END_IF;
   IF "Data_block_1".K1 AND "Data_block_1".K_B THEN "Data_block_1".ResetCounterDataSensor := TRUE; END_IF;
END_REGION

REGION Network 4: Reset Counter Data Sensor (reset) kanan ke kiri
   "IEC_Timer_0_DB_9".TON(IN := "Data_block_1".ResetCounterDataSensor AND NOT "Data_block_1".K1, PT := T#20ms);
   IF "IEC_Timer_0_DB_9".Q THEN "Data_block_1".ResetCounterDataSensor := FALSE; END_IF;
   "Data_block_1".Reset_data_baru1 := "IEC_Timer_0_DB_9".Q;
END_REGION

REGION Network 5: reset data_baru (kanan ke kiri) data_baru1
   // ketika reset aktif 
   // 
   // - maka datasuhu, array data suhu roda akan kembali 0
   // - maka counter genap kembali 0
   // - maka counter ganjil menjadi -1
   // - maka sarana akan kosong
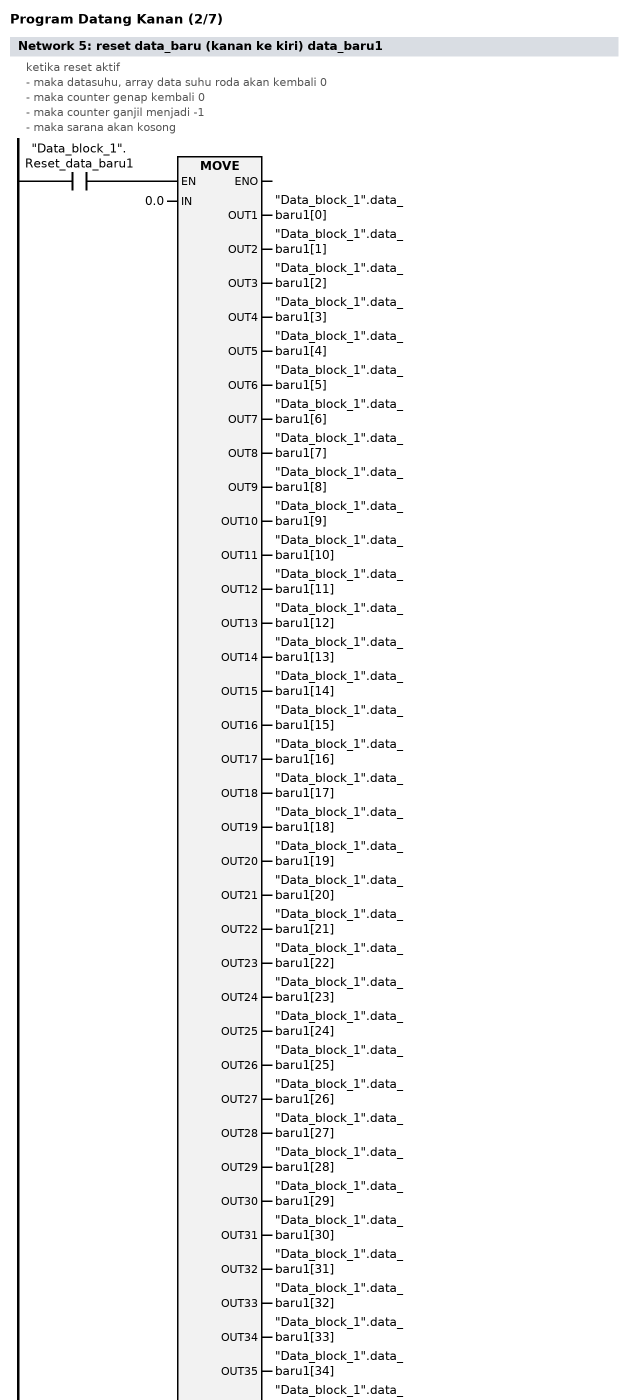
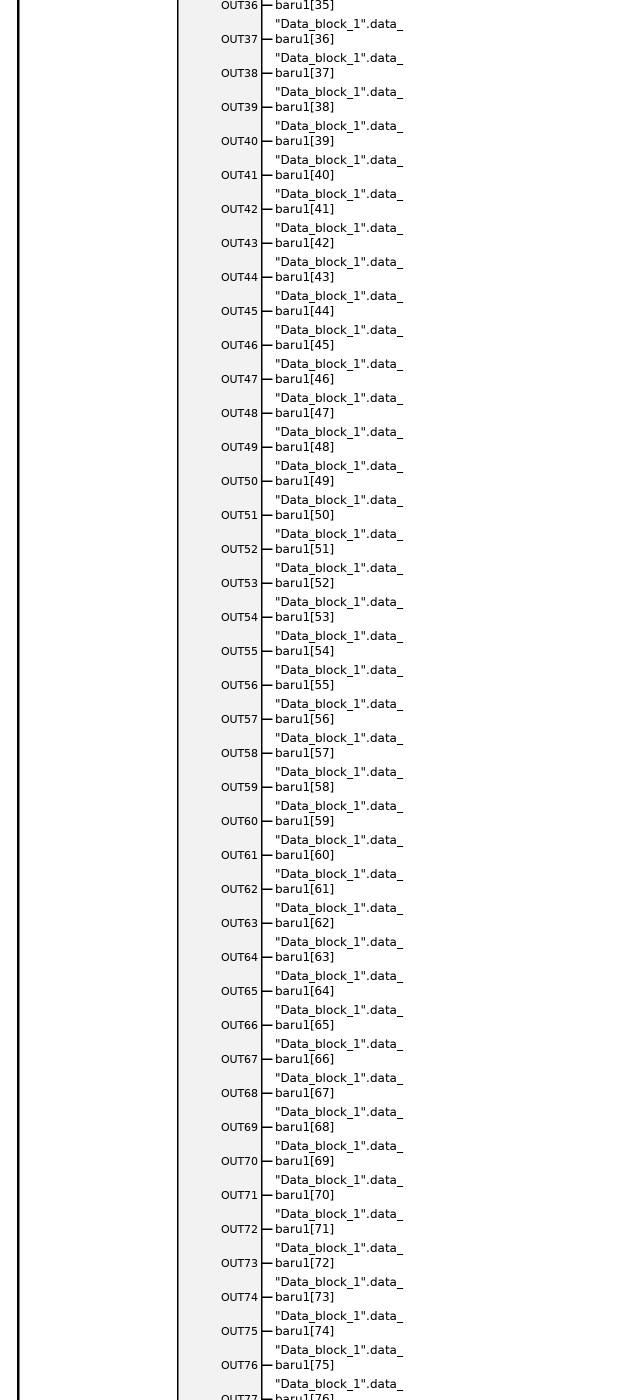
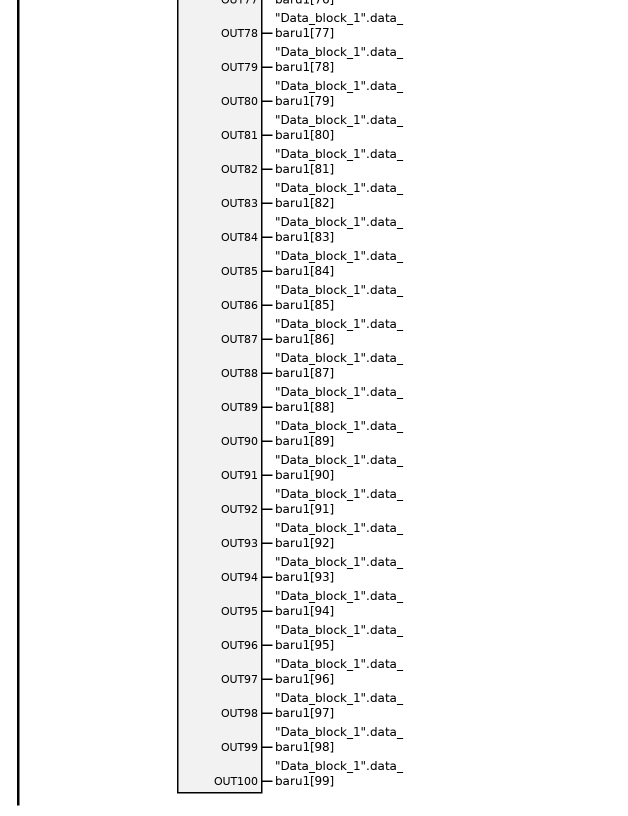
   RUNG wire#powerrail
      Contact( "Data_block_1".Reset_data_baru1 )
      Move(in := 0.0, out1 => "Data_block_1".data_baru1[0], out2 => "Data_block_1".data_baru1[1], out3 => "Data_block_1".data_baru1[2], out4 => "Data_block_1".data_baru1[3], out5 => "Data_block_1".data_baru1[4], out6 => "Data_block_1".data_baru1[5], out7 => "Data_block_1".data_baru1[6], out8 => "Data_block_1".data_baru1[7], out9 => "Data_block_1".data_baru1[8], out10 => "Data_block_1".data_baru1[9], out11 => "Data_block_1".data_baru1[10], out12 => "Data_block_1".data_baru1[11], out13 => "Data_block_1".data_baru1[12], out14 => "Data_block_1".data_baru1[13], out15 => "Data_block_1".data_baru1[14], out16 => "Data_block_1".data_baru1[15], out17 => "Data_block_1".data_baru1[16], out18 => "Data_block_1".data_baru1[17], out19 => "Data_block_1".data_baru1[18], out20 => "Data_block_1".data_baru1[19], out21 => "Data_block_1".data_baru1[20], out22 => "Data_block_1".data_baru1[21], out23 => "Data_block_1".data_baru1[22], out24 => "Data_block_1".data_baru1[23], out25 => "Data_block_1".data_baru1[24], out26 => "Data_block_1".data_baru1[25], out27 => "Data_block_1".data_baru1[26], out28 => "Data_block_1".data_baru1[27], out29 => "Data_block_1".data_baru1[28], out30 => "Data_block_1".data_baru1[29], out31 => "Data_block_1".data_baru1[30], out32 => "Data_block_1".data_baru1[31], out33 => "Data_block_1".data_baru1[32], out34 => "Data_block_1".data_baru1[33], out35 => "Data_block_1".data_baru1[34], out36 => "Data_block_1".data_baru1[35], out37 => "Data_block_1".data_baru1[36], out38 => "Data_block_1".data_baru1[37], out39 => "Data_block_1".data_baru1[38], out40 => "Data_block_1".data_baru1[39], out41 => "Data_block_1".data_baru1[40], out42 => "Data_block_1".data_baru1[41], out43 => "Data_block_1".data_baru1[42], out44 => "Data_block_1".data_baru1[43], out45 => "Data_block_1".data_baru1[44], out46 => "Data_block_1".data_baru1[45], out47 => "Data_block_1".data_baru1[46], out48 => "Data_block_1".data_baru1[47], out49 => "Data_block_1".data_baru1[48], out50 => "Data_block_1".data_baru1[49], out51 => "Data_block_1".data_baru1[50], out52 => "Data_block_1".data_baru1[51], out53 => "Data_block_1".data_baru1[52], out54 => "Data_block_1".data_baru1[53], out55 => "Data_block_1".data_baru1[54], out56 => "Data_block_1".data_baru1[55], out57 => "Data_block_1".data_baru1[56], out58 => "Data_block_1".data_baru1[57], out59 => "Data_block_1".data_baru1[58], out60 => "Data_block_1".data_baru1[59], out61 => "Data_block_1".data_baru1[60], out62 => "Data_block_1".data_baru1[61], out63 => "Data_block_1".data_baru1[62], out64 => "Data_block_1".data_baru1[63], out65 => "Data_block_1".data_baru1[64], out66 => "Data_block_1".data_baru1[65], out67 => "Data_block_1".data_baru1[66], out68 => "Data_block_1".data_baru1[67], out69 => "Data_block_1".data_baru1[68], out70 => "Data_block_1".data_baru1[69], out71 => "Data_block_1".data_baru1[70], out72 => "Data_block_1".data_baru1[71], out73 => "Data_block_1".data_baru1[72], out74 => "Data_block_1".data_baru1[73], out75 => "Data_block_1".data_baru1[74], out76 => "Data_block_1".data_baru1[75], out77 => "Data_block_1".data_baru1[76], out78 => "Data_block_1".data_baru1[77], out79 => "Data_block_1".data_baru1[78], out80 => "Data_block_1".data_baru1[79], out81 => "Data_block_1".data_baru1[80], out82 => "Data_block_1".data_baru1[81], out83 => "Data_block_1".data_baru1[82], out84 => "Data_block_1".data_baru1[83], out85 => "Data_block_1".data_baru1[84], out86 => "Data_block_1".data_baru1[85], out87 => "Data_block_1".data_baru1[86], out88 => "Data_block_1".data_baru1[87], out89 => "Data_block_1".data_baru1[88], out90 => "Data_block_1".data_baru1[89], out91 => "Data_block_1".data_baru1[90], out92 => "Data_block_1".data_baru1[91], out93 => "Data_block_1".data_baru1[92], out94 => "Data_block_1".data_baru1[93], out95 => "Data_block_1".data_baru1[94], out96 => "Data_block_1".data_baru1[95], out97 => "Data_block_1".data_baru1[96], out98 => "Data_block_1".data_baru1[97], out99 => "Data_block_1".data_baru1[98], out100 => "Data_block_1".data_baru1[99])
   END_RUNG
   // the same network as SCL:
   IF "Data_block_1".Reset_data_baru1 THEN
       "Data_block_1".data_baru1[0] := 0.0;
       "Data_block_1".data_baru1[1] := 0.0;
       "Data_block_1".data_baru1[2] := 0.0;
       "Data_block_1".data_baru1[3] := 0.0;
       "Data_block_1".data_baru1[4] := 0.0;
       "Data_block_1".data_baru1[5] := 0.0;
       "Data_block_1".data_baru1[6] := 0.0;
       "Data_block_1".data_baru1[7] := 0.0;
       "Data_block_1".data_baru1[8] := 0.0;
       "Data_block_1".data_baru1[9] := 0.0;
       "Data_block_1".data_baru1[10] := 0.0;
       "Data_block_1".data_baru1[11] := 0.0;
       "Data_block_1".data_baru1[12] := 0.0;
       "Data_block_1".data_baru1[13] := 0.0;
       "Data_block_1".data_baru1[14] := 0.0;
       "Data_block_1".data_baru1[15] := 0.0;
       "Data_block_1".data_baru1[16] := 0.0;
       "Data_block_1".data_baru1[17] := 0.0;
       "Data_block_1".data_baru1[18] := 0.0;
       "Data_block_1".data_baru1[19] := 0.0;
       "Data_block_1".data_baru1[20] := 0.0;
       "Data_block_1".data_baru1[21] := 0.0;
       "Data_block_1".data_baru1[22] := 0.0;
       "Data_block_1".data_baru1[23] := 0.0;
       "Data_block_1".data_baru1[24] := 0.0;
       "Data_block_1".data_baru1[25] := 0.0;
       "Data_block_1".data_baru1[26] := 0.0;
       "Data_block_1".data_baru1[27] := 0.0;
       "Data_block_1".data_baru1[28] := 0.0;
       "Data_block_1".data_baru1[29] := 0.0;
       "Data_block_1".data_baru1[30] := 0.0;
       "Data_block_1".data_baru1[31] := 0.0;
       "Data_block_1".data_baru1[32] := 0.0;
       "Data_block_1".data_baru1[33] := 0.0;
       "Data_block_1".data_baru1[34] := 0.0;
       "Data_block_1".data_baru1[35] := 0.0;
       "Data_block_1".data_baru1[36] := 0.0;
       "Data_block_1".data_baru1[37] := 0.0;
       "Data_block_1".data_baru1[38] := 0.0;
       "Data_block_1".data_baru1[39] := 0.0;
       "Data_block_1".data_baru1[40] := 0.0;
       "Data_block_1".data_baru1[41] := 0.0;
       "Data_block_1".data_baru1[42] := 0.0;
       "Data_block_1".data_baru1[43] := 0.0;
       "Data_block_1".data_baru1[44] := 0.0;
       "Data_block_1".data_baru1[45] := 0.0;
       "Data_block_1".data_baru1[46] := 0.0;
       "Data_block_1".data_baru1[47] := 0.0;
       "Data_block_1".data_baru1[48] := 0.0;
       "Data_block_1".data_baru1[49] := 0.0;
       "Data_block_1".data_baru1[50] := 0.0;
       "Data_block_1".data_baru1[51] := 0.0;
       "Data_block_1".data_baru1[52] := 0.0;
       "Data_block_1".data_baru1[53] := 0.0;
       "Data_block_1".data_baru1[54] := 0.0;
       "Data_block_1".data_baru1[55] := 0.0;
       "Data_block_1".data_baru1[56] := 0.0;
       "Data_block_1".data_baru1[57] := 0.0;
       "Data_block_1".data_baru1[58] := 0.0;
       "Data_block_1".data_baru1[59] := 0.0;
       "Data_block_1".data_baru1[60] := 0.0;
       "Data_block_1".data_baru1[61] := 0.0;
       "Data_block_1".data_baru1[62] := 0.0;
       "Data_block_1".data_baru1[63] := 0.0;
       "Data_block_1".data_baru1[64] := 0.0;
       "Data_block_1".data_baru1[65] := 0.0;
       "Data_block_1".data_baru1[66] := 0.0;
       "Data_block_1".data_baru1[67] := 0.0;
       "Data_block_1".data_baru1[68] := 0.0;
       "Data_block_1".data_baru1[69] := 0.0;
       "Data_block_1".data_baru1[70] := 0.0;
       "Data_block_1".data_baru1[71] := 0.0;
       "Data_block_1".data_baru1[72] := 0.0;
       "Data_block_1".data_baru1[73] := 0.0;
       "Data_block_1".data_baru1[74] := 0.0;
       "Data_block_1".data_baru1[75] := 0.0;
       "Data_block_1".data_baru1[76] := 0.0;
       "Data_block_1".data_baru1[77] := 0.0;
       "Data_block_1".data_baru1[78] := 0.0;
       "Data_block_1".data_baru1[79] := 0.0;
       "Data_block_1".data_baru1[80] := 0.0;
       "Data_block_1".data_baru1[81] := 0.0;
       "Data_block_1".data_baru1[82] := 0.0;
       "Data_block_1".data_baru1[83] := 0.0;
       "Data_block_1".data_baru1[84] := 0.0;
       "Data_block_1".data_baru1[85] := 0.0;
       "Data_block_1".data_baru1[86] := 0.0;
       "Data_block_1".data_baru1[87] := 0.0;
       "Data_block_1".data_baru1[88] := 0.0;
       "Data_block_1".data_baru1[89] := 0.0;
       "Data_block_1".data_baru1[90] := 0.0;
       "Data_block_1".data_baru1[91] := 0.0;
       "Data_block_1".data_baru1[92] := 0.0;
       "Data_block_1".data_baru1[93] := 0.0;
       "Data_block_1".data_baru1[94] := 0.0;
       "Data_block_1".data_baru1[95] := 0.0;
       "Data_block_1".data_baru1[96] := 0.0;
       "Data_block_1".data_baru1[97] := 0.0;
       "Data_block_1".data_baru1[98] := 0.0;
       "Data_block_1".data_baru1[99] := 0.0;
   END_IF;
END_REGION

REGION Network 6: Koil Set Proxy A (kanan ke kiri)
   // Sensor A aktif, menunjukkan arah kereta dari arah kanan
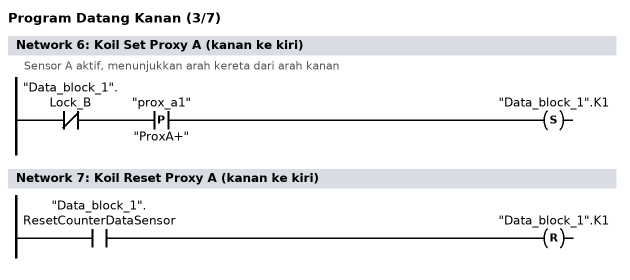
   RUNG wire#powerrail
      I_Contact( "Data_block_1".Lock_B )
      P_Contact(operand := "prox_a1", bit := "ProxA+")
      S_Coil( "Data_block_1".K1 )
   END_RUNG
   // the same network as SCL:
   #_w1 := NOT "Data_block_1".Lock_B AND "prox_a1" AND NOT "ProxA+";   // rising edge of "prox_a1"
   "ProxA+" := "prox_a1";
   IF #_w1 THEN "Data_block_1".K1 := TRUE; END_IF;
END_REGION

REGION Network 7: Koil Reset Proxy A (kanan ke kiri)
   RUNG wire#powerrail
      Contact( "Data_block_1".ResetCounterDataSensor )
      R_Coil( "Data_block_1".K1 )
   END_RUNG
   // the same network as SCL:
   IF "Data_block_1".ResetCounterDataSensor THEN "Data_block_1".K1 := FALSE; END_IF;
END_REGION

REGION Network 8: Mengukur Suhu Roda (kanan ke kiri) Data_baru1
   // setelah sensor suhu aktif membaca
   // kemudian counter menghitung jumlah berapa kali sensor suhu mendeteksi suhu pada satu roda
   // 
   // apabila data sensor suhu yang terbaca(datasensor) tidak sama dengan nol maka data suhu yang terbaca(datasensor) dipindahkan ke array data suhu baru (data_baru1 untuk sebelah kanan) (data_baru2 untuk sebelah kiri)
   // data sensor terbaru dirubah jadi data baru
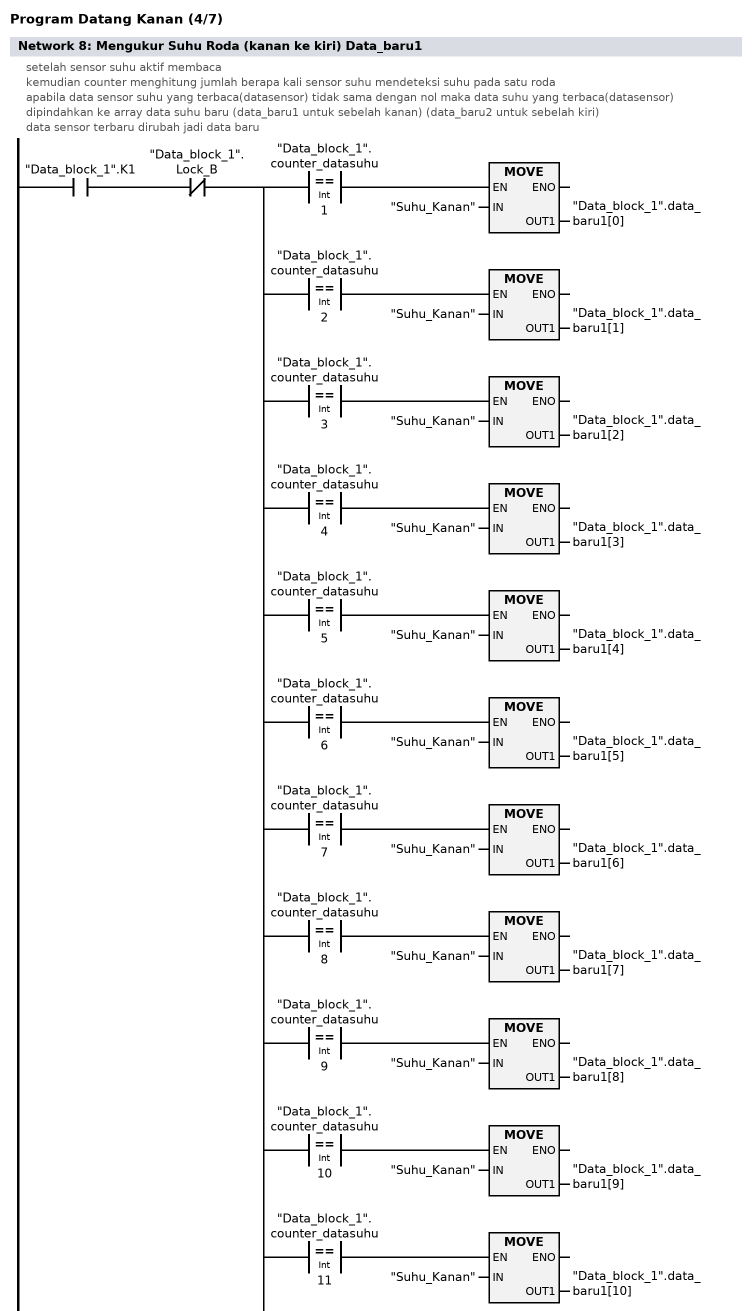
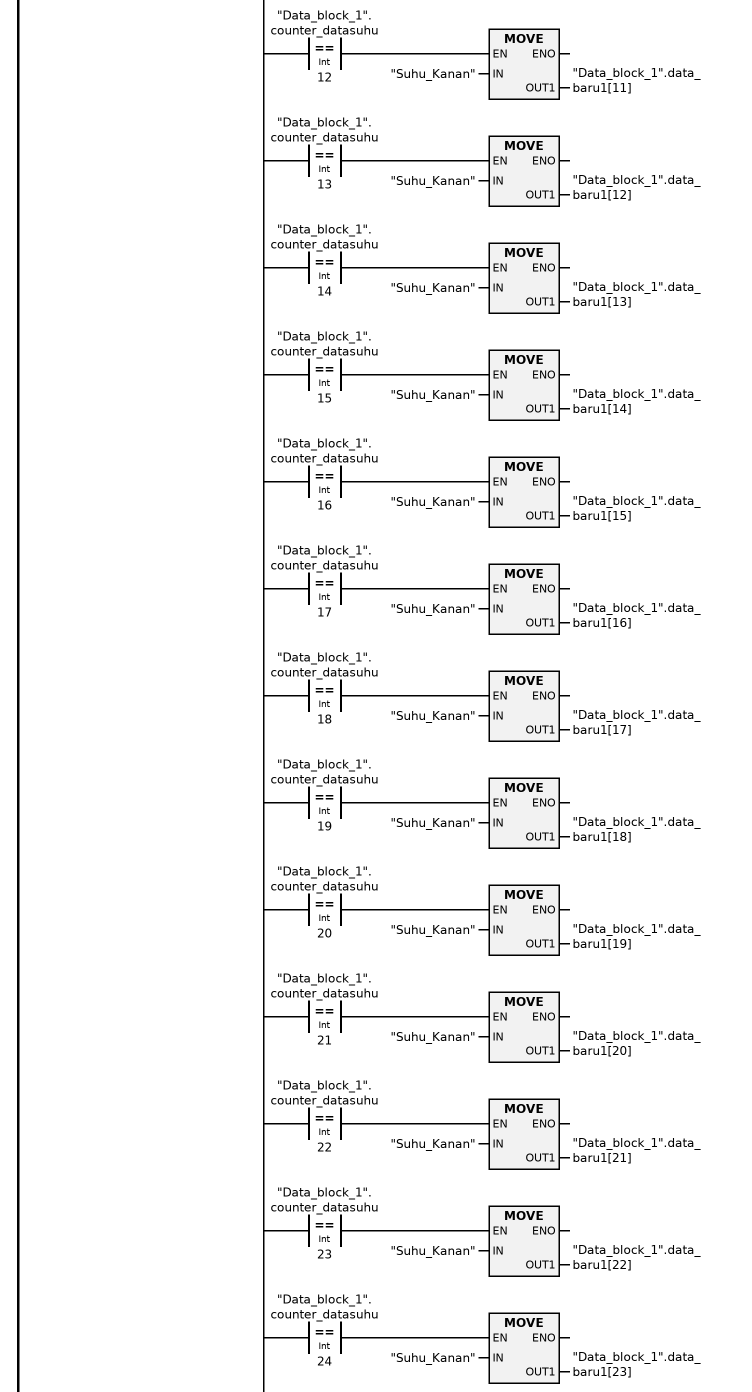
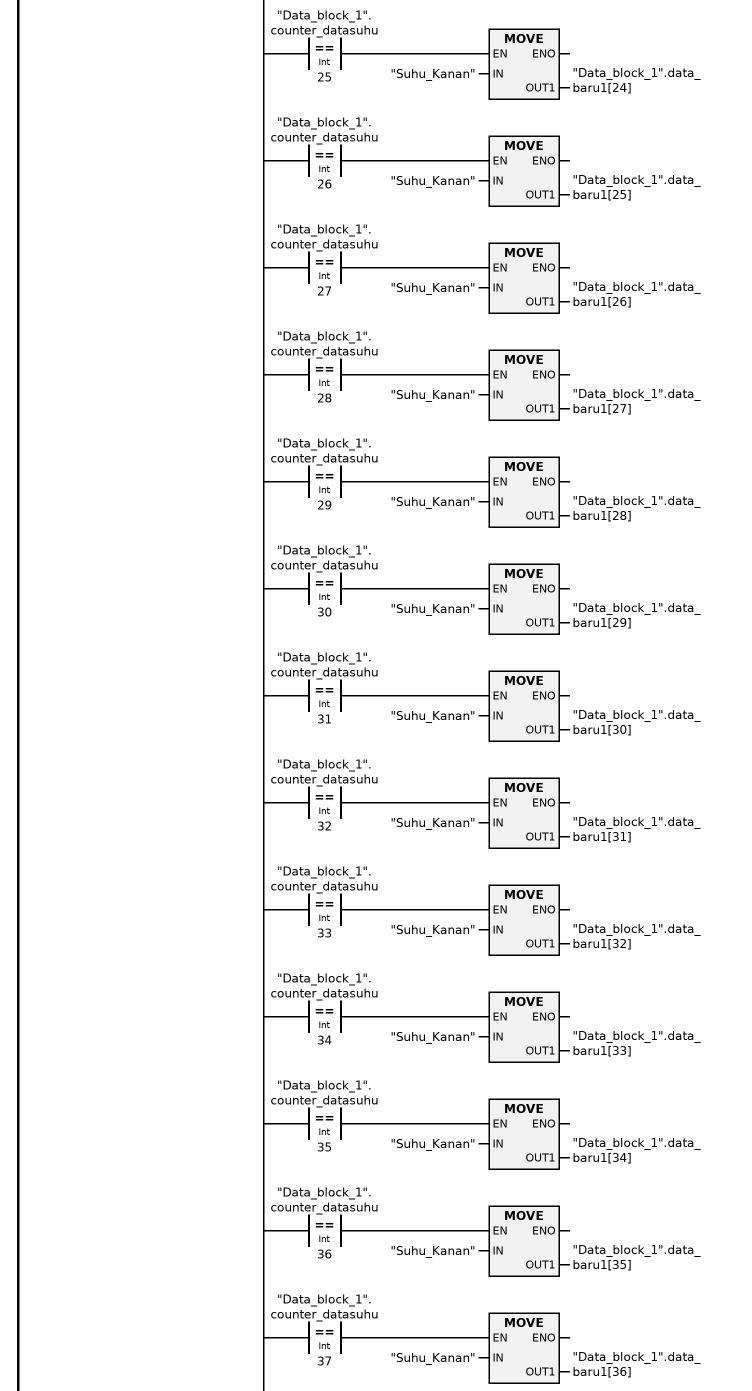
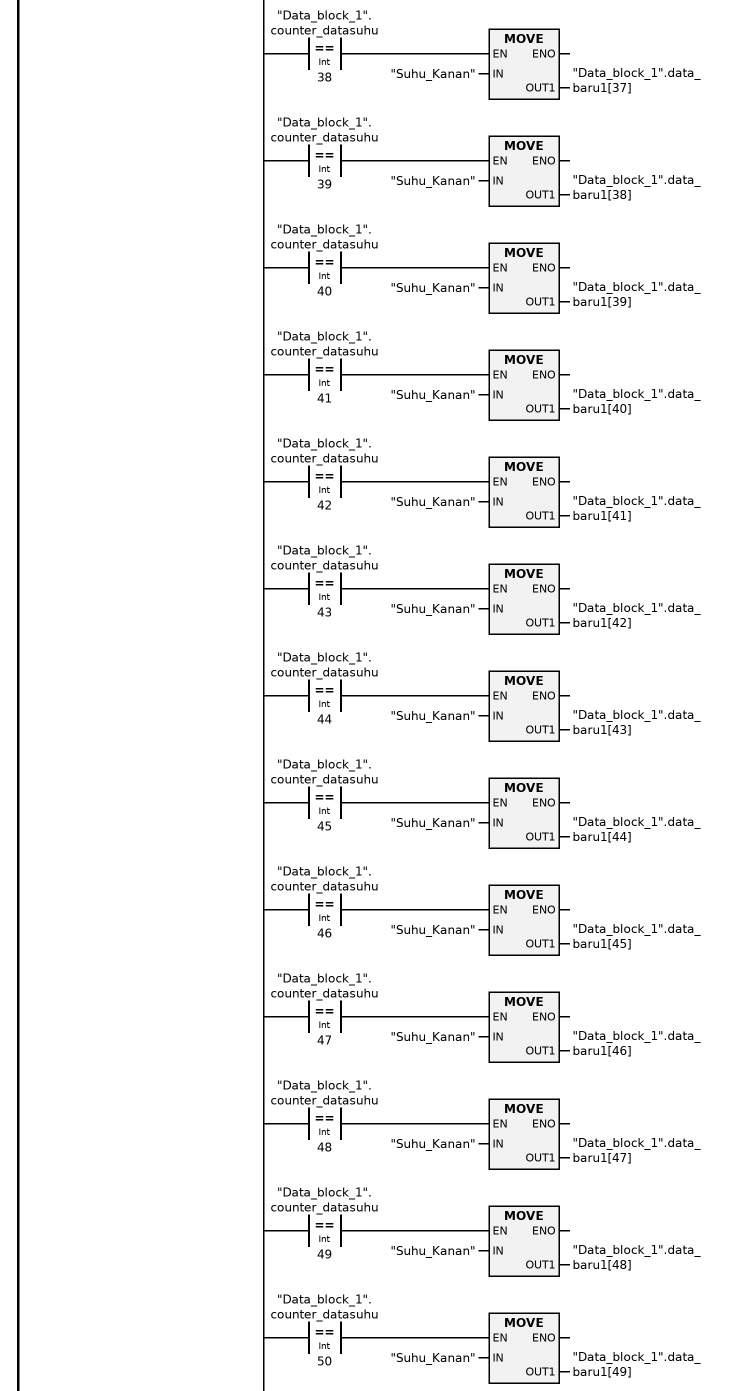
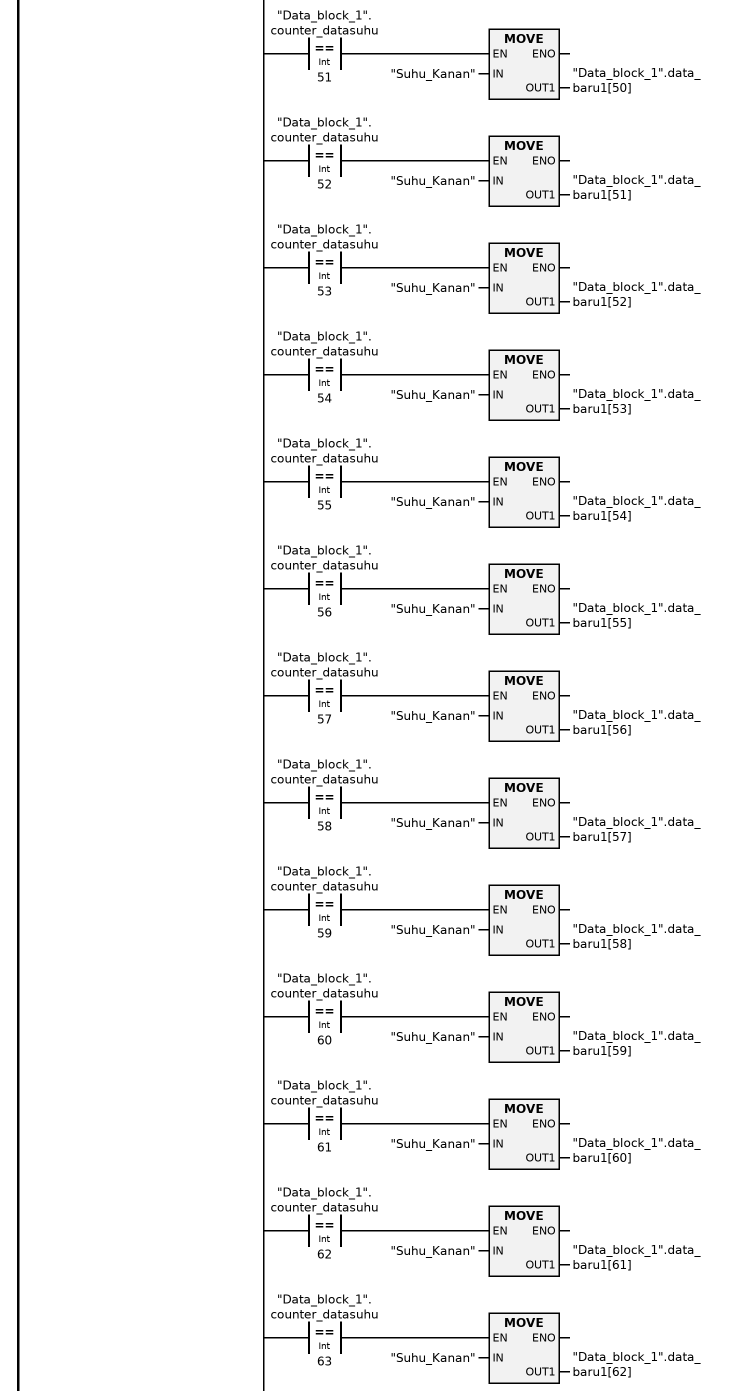
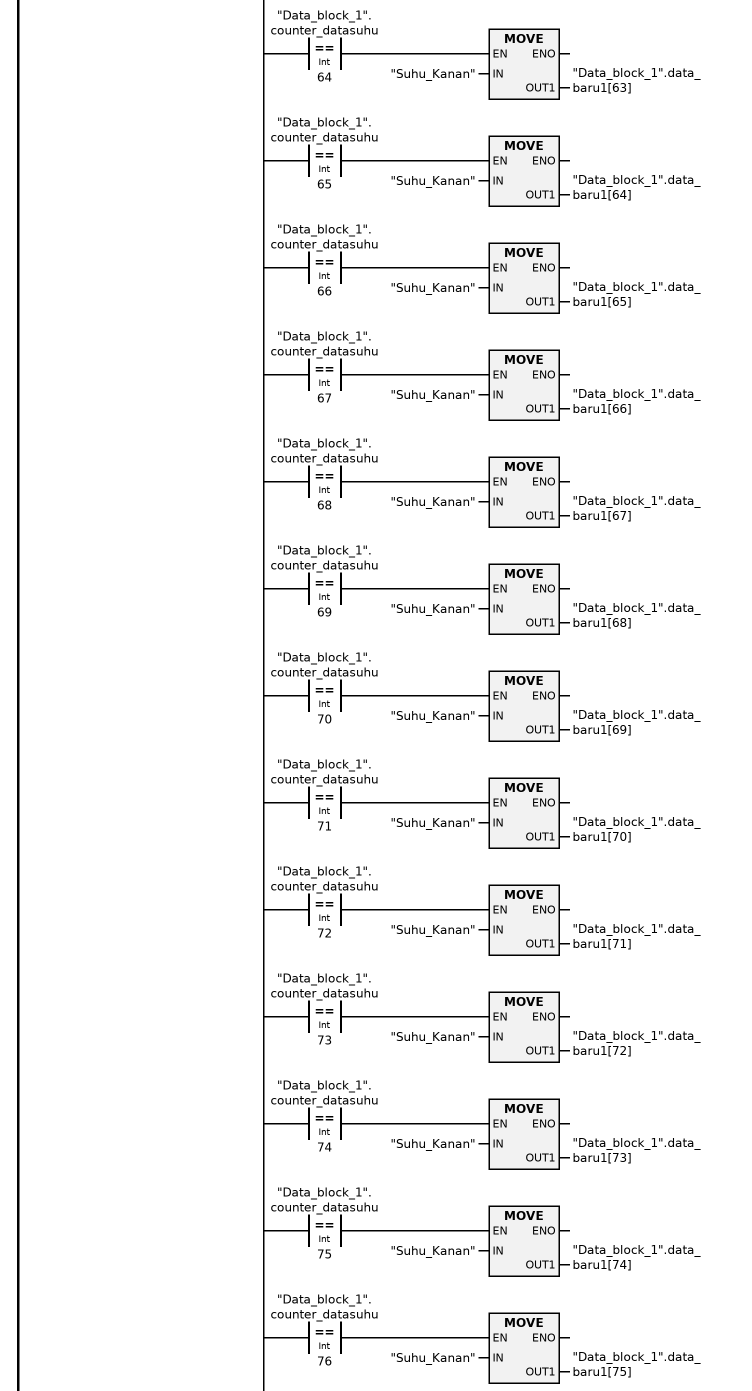
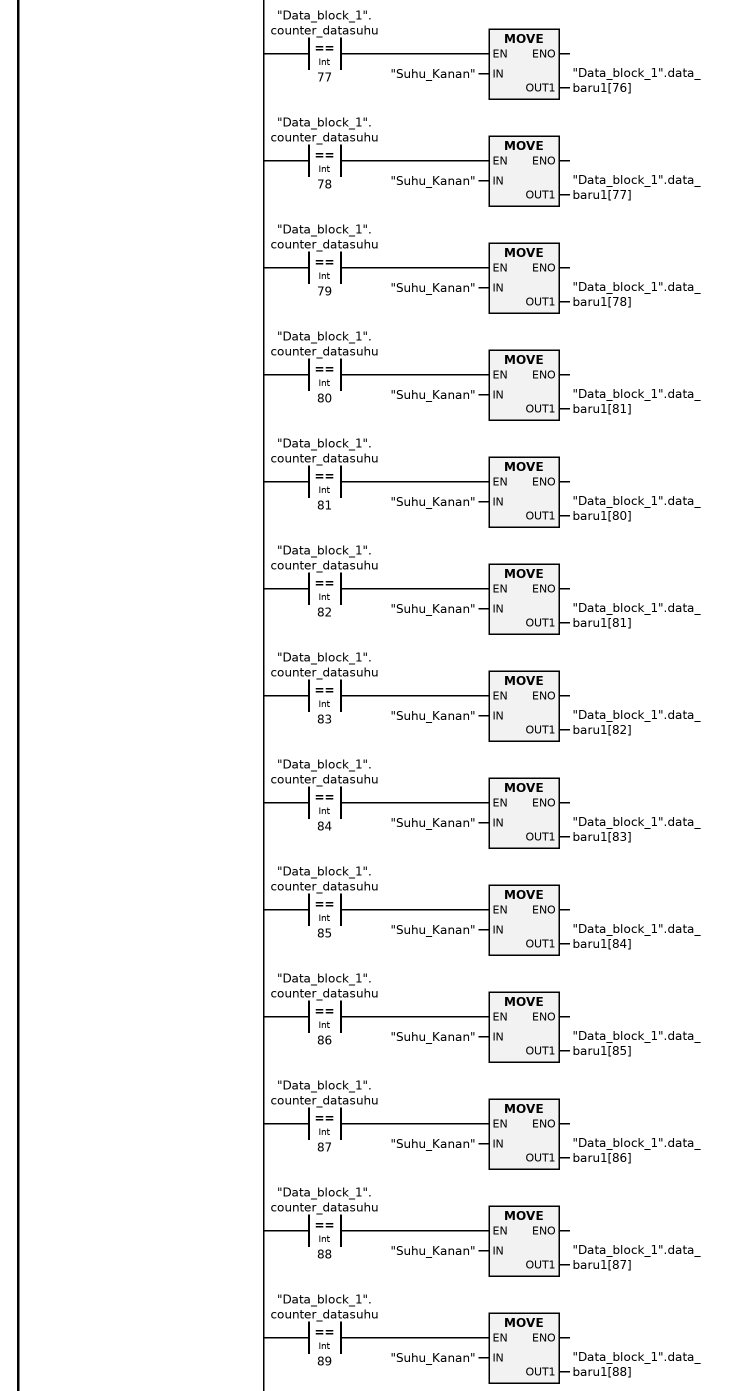
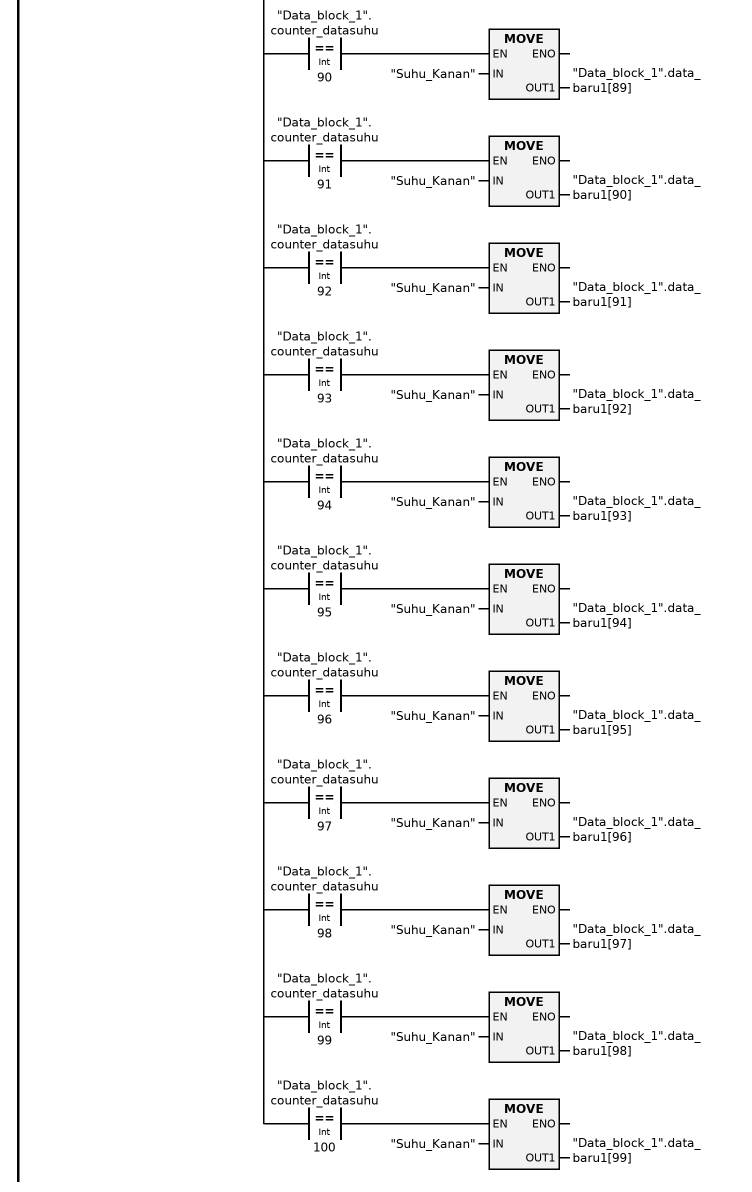
   RUNG wire#powerrail
      Contact( "Data_block_1".K1 )
      I_Contact( "Data_block_1".Lock_B )
      wire#w1
      { S7_Templates := "SrcType := Int" } EQ_Contact(in1 := "Data_block_1".counter_datasuhu, in2 := 1)
      Move(in := "Suhu_Kanan", out1 => "Data_block_1".data_baru1[0])
   END_RUNG
   RUNG wire#w1
      { S7_Templates := "SrcType := Int" } EQ_Contact(in1 := "Data_block_1".counter_datasuhu, in2 := 2)
      Move(in := "Suhu_Kanan", out1 => "Data_block_1".data_baru1[1])
   END_RUNG
   RUNG wire#w1
      { S7_Templates := "SrcType := Int" } EQ_Contact(in1 := "Data_block_1".counter_datasuhu, in2 := 3)
      Move(in := "Suhu_Kanan", out1 => "Data_block_1".data_baru1[2])
   END_RUNG
   RUNG wire#w1
      { S7_Templates := "SrcType := Int" } EQ_Contact(in1 := "Data_block_1".counter_datasuhu, in2 := 4)
      Move(in := "Suhu_Kanan", out1 => "Data_block_1".data_baru1[3])
   END_RUNG
   RUNG wire#w1
      { S7_Templates := "SrcType := Int" } EQ_Contact(in1 := "Data_block_1".counter_datasuhu, in2 := 5)
      Move(in := "Suhu_Kanan", out1 => "Data_block_1".data_baru1[4])
   END_RUNG
   RUNG wire#w1
      { S7_Templates := "SrcType := Int" } EQ_Contact(in1 := "Data_block_1".counter_datasuhu, in2 := 6)
      Move(in := "Suhu_Kanan", out1 => "Data_block_1".data_baru1[5])
   END_RUNG
   RUNG wire#w1
      { S7_Templates := "SrcType := Int" } EQ_Contact(in1 := "Data_block_1".counter_datasuhu, in2 := 7)
      Move(in := "Suhu_Kanan", out1 => "Data_block_1".data_baru1[6])
   END_RUNG
   RUNG wire#w1
      { S7_Templates := "SrcType := Int" } EQ_Contact(in1 := "Data_block_1".counter_datasuhu, in2 := 8)
      Move(in := "Suhu_Kanan", out1 => "Data_block_1".data_baru1[7])
   END_RUNG
   RUNG wire#w1
      { S7_Templates := "SrcType := Int" } EQ_Contact(in1 := "Data_block_1".counter_datasuhu, in2 := 9)
      Move(in := "Suhu_Kanan", out1 => "Data_block_1".data_baru1[8])
   END_RUNG
   RUNG wire#w1
      { S7_Templates := "SrcType := Int" } EQ_Contact(in1 := "Data_block_1".counter_datasuhu, in2 := 10)
      Move(in := "Suhu_Kanan", out1 => "Data_block_1".data_baru1[9])
   END_RUNG
   RUNG wire#w1
      { S7_Templates := "SrcType := Int" } EQ_Contact(in1 := "Data_block_1".counter_datasuhu, in2 := 11)
      Move(in := "Suhu_Kanan", out1 => "Data_block_1".data_baru1[10])
   END_RUNG
   RUNG wire#w1
      { S7_Templates := "SrcType := Int" } EQ_Contact(in1 := "Data_block_1".counter_datasuhu, in2 := 12)
      Move(in := "Suhu_Kanan", out1 => "Data_block_1".data_baru1[11])
   END_RUNG
   RUNG wire#w1
      { S7_Templates := "SrcType := Int" } EQ_Contact(in1 := "Data_block_1".counter_datasuhu, in2 := 13)
      Move(in := "Suhu_Kanan", out1 => "Data_block_1".data_baru1[12])
   END_RUNG
   RUNG wire#w1
      { S7_Templates := "SrcType := Int" } EQ_Contact(in1 := "Data_block_1".counter_datasuhu, in2 := 14)
      Move(in := "Suhu_Kanan", out1 => "Data_block_1".data_baru1[13])
   END_RUNG
   RUNG wire#w1
      { S7_Templates := "SrcType := Int" } EQ_Contact(in1 := "Data_block_1".counter_datasuhu, in2 := 15)
      Move(in := "Suhu_Kanan", out1 => "Data_block_1".data_baru1[14])
   END_RUNG
   RUNG wire#w1
      { S7_Templates := "SrcType := Int" } EQ_Contact(in1 := "Data_block_1".counter_datasuhu, in2 := 16)
      Move(in := "Suhu_Kanan", out1 => "Data_block_1".data_baru1[15])
   END_RUNG
   RUNG wire#w1
      { S7_Templates := "SrcType := Int" } EQ_Contact(in1 := "Data_block_1".counter_datasuhu, in2 := 17)
      Move(in := "Suhu_Kanan", out1 => "Data_block_1".data_baru1[16])
   END_RUNG
   RUNG wire#w1
      { S7_Templates := "SrcType := Int" } EQ_Contact(in1 := "Data_block_1".counter_datasuhu, in2 := 18)
      Move(in := "Suhu_Kanan", out1 => "Data_block_1".data_baru1[17])
   END_RUNG
   RUNG wire#w1
      { S7_Templates := "SrcType := Int" } EQ_Contact(in1 := "Data_block_1".counter_datasuhu, in2 := 19)
      Move(in := "Suhu_Kanan", out1 => "Data_block_1".data_baru1[18])
   END_RUNG
   RUNG wire#w1
      { S7_Templates := "SrcType := Int" } EQ_Contact(in1 := "Data_block_1".counter_datasuhu, in2 := 20)
      Move(in := "Suhu_Kanan", out1 => "Data_block_1".data_baru1[19])
   END_RUNG
   RUNG wire#w1
      { S7_Templates := "SrcType := Int" } EQ_Contact(in1 := "Data_block_1".counter_datasuhu, in2 := 21)
      Move(in := "Suhu_Kanan", out1 => "Data_block_1".data_baru1[20])
   END_RUNG
   RUNG wire#w1
      { S7_Templates := "SrcType := Int" } EQ_Contact(in1 := "Data_block_1".counter_datasuhu, in2 := 22)
      Move(in := "Suhu_Kanan", out1 => "Data_block_1".data_baru1[21])
   END_RUNG
   RUNG wire#w1
      { S7_Templates := "SrcType := Int" } EQ_Contact(in1 := "Data_block_1".counter_datasuhu, in2 := 23)
      Move(in := "Suhu_Kanan", out1 => "Data_block_1".data_baru1[22])
   END_RUNG
   RUNG wire#w1
      { S7_Templates := "SrcType := Int" } EQ_Contact(in1 := "Data_block_1".counter_datasuhu, in2 := 24)
      Move(in := "Suhu_Kanan", out1 => "Data_block_1".data_baru1[23])
   END_RUNG
   RUNG wire#w1
      { S7_Templates := "SrcType := Int" } EQ_Contact(in1 := "Data_block_1".counter_datasuhu, in2 := 25)
      Move(in := "Suhu_Kanan", out1 => "Data_block_1".data_baru1[24])
   END_RUNG
   RUNG wire#w1
      { S7_Templates := "SrcType := Int" } EQ_Contact(in1 := "Data_block_1".counter_datasuhu, in2 := 26)
      Move(in := "Suhu_Kanan", out1 => "Data_block_1".data_baru1[25])
   END_RUNG
   RUNG wire#w1
      { S7_Templates := "SrcType := Int" } EQ_Contact(in1 := "Data_block_1".counter_datasuhu, in2 := 27)
      Move(in := "Suhu_Kanan", out1 => "Data_block_1".data_baru1[26])
   END_RUNG
   RUNG wire#w1
      { S7_Templates := "SrcType := Int" } EQ_Contact(in1 := "Data_block_1".counter_datasuhu, in2 := 28)
      Move(in := "Suhu_Kanan", out1 => "Data_block_1".data_baru1[27])
   END_RUNG
   RUNG wire#w1
      { S7_Templates := "SrcType := Int" } EQ_Contact(in1 := "Data_block_1".counter_datasuhu, in2 := 29)
      Move(in := "Suhu_Kanan", out1 => "Data_block_1".data_baru1[28])
   END_RUNG
   RUNG wire#w1
      { S7_Templates := "SrcType := Int" } EQ_Contact(in1 := "Data_block_1".counter_datasuhu, in2 := 30)
      Move(in := "Suhu_Kanan", out1 => "Data_block_1".data_baru1[29])
   END_RUNG
   RUNG wire#w1
      { S7_Templates := "SrcType := Int" } EQ_Contact(in1 := "Data_block_1".counter_datasuhu, in2 := 31)
      Move(in := "Suhu_Kanan", out1 => "Data_block_1".data_baru1[30])
   END_RUNG
   RUNG wire#w1
      { S7_Templates := "SrcType := Int" } EQ_Contact(in1 := "Data_block_1".counter_datasuhu, in2 := 32)
      Move(in := "Suhu_Kanan", out1 => "Data_block_1".data_baru1[31])
   END_RUNG
   RUNG wire#w1
      { S7_Templates := "SrcType := Int" } EQ_Contact(in1 := "Data_block_1".counter_datasuhu, in2 := 33)
      Move(in := "Suhu_Kanan", out1 => "Data_block_1".data_baru1[32])
   END_RUNG
   RUNG wire#w1
      { S7_Templates := "SrcType := Int" } EQ_Contact(in1 := "Data_block_1".counter_datasuhu, in2 := 34)
      Move(in := "Suhu_Kanan", out1 => "Data_block_1".data_baru1[33])
   END_RUNG
   RUNG wire#w1
      { S7_Templates := "SrcType := Int" } EQ_Contact(in1 := "Data_block_1".counter_datasuhu, in2 := 35)
      Move(in := "Suhu_Kanan", out1 => "Data_block_1".data_baru1[34])
   END_RUNG
   RUNG wire#w1
      { S7_Templates := "SrcType := Int" } EQ_Contact(in1 := "Data_block_1".counter_datasuhu, in2 := 36)
      Move(in := "Suhu_Kanan", out1 => "Data_block_1".data_baru1[35])
   END_RUNG
   RUNG wire#w1
      { S7_Templates := "SrcType := Int" } EQ_Contact(in1 := "Data_block_1".counter_datasuhu, in2 := 37)
      Move(in := "Suhu_Kanan", out1 => "Data_block_1".data_baru1[36])
   END_RUNG
   RUNG wire#w1
      { S7_Templates := "SrcType := Int" } EQ_Contact(in1 := "Data_block_1".counter_datasuhu, in2 := 38)
      Move(in := "Suhu_Kanan", out1 => "Data_block_1".data_baru1[37])
   END_RUNG
   RUNG wire#w1
      { S7_Templates := "SrcType := Int" } EQ_Contact(in1 := "Data_block_1".counter_datasuhu, in2 := 39)
      Move(in := "Suhu_Kanan", out1 => "Data_block_1".data_baru1[38])
   END_RUNG
   RUNG wire#w1
      { S7_Templates := "SrcType := Int" } EQ_Contact(in1 := "Data_block_1".counter_datasuhu, in2 := 40)
      Move(in := "Suhu_Kanan", out1 => "Data_block_1".data_baru1[39])
   END_RUNG
   RUNG wire#w1
      { S7_Templates := "SrcType := Int" } EQ_Contact(in1 := "Data_block_1".counter_datasuhu, in2 := 41)
      Move(in := "Suhu_Kanan", out1 => "Data_block_1".data_baru1[40])
   END_RUNG
   RUNG wire#w1
      { S7_Templates := "SrcType := Int" } EQ_Contact(in1 := "Data_block_1".counter_datasuhu, in2 := 42)
      Move(in := "Suhu_Kanan", out1 => "Data_block_1".data_baru1[41])
   END_RUNG
   RUNG wire#w1
      { S7_Templates := "SrcType := Int" } EQ_Contact(in1 := "Data_block_1".counter_datasuhu, in2 := 43)
      Move(in := "Suhu_Kanan", out1 => "Data_block_1".data_baru1[42])
   END_RUNG
   RUNG wire#w1
      { S7_Templates := "SrcType := Int" } EQ_Contact(in1 := "Data_block_1".counter_datasuhu, in2 := 44)
      Move(in := "Suhu_Kanan", out1 => "Data_block_1".data_baru1[43])
   END_RUNG
   RUNG wire#w1
      { S7_Templates := "SrcType := Int" } EQ_Contact(in1 := "Data_block_1".counter_datasuhu, in2 := 45)
      Move(in := "Suhu_Kanan", out1 => "Data_block_1".data_baru1[44])
   END_RUNG
   RUNG wire#w1
      { S7_Templates := "SrcType := Int" } EQ_Contact(in1 := "Data_block_1".counter_datasuhu, in2 := 46)
      Move(in := "Suhu_Kanan", out1 => "Data_block_1".data_baru1[45])
   END_RUNG
   RUNG wire#w1
      { S7_Templates := "SrcType := Int" } EQ_Contact(in1 := "Data_block_1".counter_datasuhu, in2 := 47)
      Move(in := "Suhu_Kanan", out1 => "Data_block_1".data_baru1[46])
   END_RUNG
   RUNG wire#w1
      { S7_Templates := "SrcType := Int" } EQ_Contact(in1 := "Data_block_1".counter_datasuhu, in2 := 48)
      Move(in := "Suhu_Kanan", out1 => "Data_block_1".data_baru1[47])
   END_RUNG
   RUNG wire#w1
      { S7_Templates := "SrcType := Int" } EQ_Contact(in1 := "Data_block_1".counter_datasuhu, in2 := 49)
      Move(in := "Suhu_Kanan", out1 => "Data_block_1".data_baru1[48])
   END_RUNG
   RUNG wire#w1
      { S7_Templates := "SrcType := Int" } EQ_Contact(in1 := "Data_block_1".counter_datasuhu, in2 := 50)
      Move(in := "Suhu_Kanan", out1 => "Data_block_1".data_baru1[49])
   END_RUNG
   RUNG wire#w1
      { S7_Templates := "SrcType := Int" } EQ_Contact(in1 := "Data_block_1".counter_datasuhu, in2 := 51)
      Move(in := "Suhu_Kanan", out1 => "Data_block_1".data_baru1[50])
   END_RUNG
   RUNG wire#w1
      { S7_Templates := "SrcType := Int" } EQ_Contact(in1 := "Data_block_1".counter_datasuhu, in2 := 52)
      Move(in := "Suhu_Kanan", out1 => "Data_block_1".data_baru1[51])
   END_RUNG
   RUNG wire#w1
      { S7_Templates := "SrcType := Int" } EQ_Contact(in1 := "Data_block_1".counter_datasuhu, in2 := 53)
      Move(in := "Suhu_Kanan", out1 => "Data_block_1".data_baru1[52])
   END_RUNG
   RUNG wire#w1
      { S7_Templates := "SrcType := Int" } EQ_Contact(in1 := "Data_block_1".counter_datasuhu, in2 := 54)
      Move(in := "Suhu_Kanan", out1 => "Data_block_1".data_baru1[53])
   END_RUNG
   RUNG wire#w1
      { S7_Templates := "SrcType := Int" } EQ_Contact(in1 := "Data_block_1".counter_datasuhu, in2 := 55)
      Move(in := "Suhu_Kanan", out1 => "Data_block_1".data_baru1[54])
   END_RUNG
   RUNG wire#w1
      { S7_Templates := "SrcType := Int" } EQ_Contact(in1 := "Data_block_1".counter_datasuhu, in2 := 56)
      Move(in := "Suhu_Kanan", out1 => "Data_block_1".data_baru1[55])
   END_RUNG
   RUNG wire#w1
      { S7_Templates := "SrcType := Int" } EQ_Contact(in1 := "Data_block_1".counter_datasuhu, in2 := 57)
      Move(in := "Suhu_Kanan", out1 => "Data_block_1".data_baru1[56])
   END_RUNG
   RUNG wire#w1
      { S7_Templates := "SrcType := Int" } EQ_Contact(in1 := "Data_block_1".counter_datasuhu, in2 := 58)
      Move(in := "Suhu_Kanan", out1 => "Data_block_1".data_baru1[57])
   END_RUNG
   RUNG wire#w1
      { S7_Templates := "SrcType := Int" } EQ_Contact(in1 := "Data_block_1".counter_datasuhu, in2 := 59)
      Move(in := "Suhu_Kanan", out1 => "Data_block_1".data_baru1[58])
   END_RUNG
   RUNG wire#w1
      { S7_Templates := "SrcType := Int" } EQ_Contact(in1 := "Data_block_1".counter_datasuhu, in2 := 60)
      Move(in := "Suhu_Kanan", out1 => "Data_block_1".data_baru1[59])
   END_RUNG
   RUNG wire#w1
      { S7_Templates := "SrcType := Int" } EQ_Contact(in1 := "Data_block_1".counter_datasuhu, in2 := 61)
      Move(in := "Suhu_Kanan", out1 => "Data_block_1".data_baru1[60])
   END_RUNG
   RUNG wire#w1
      { S7_Templates := "SrcType := Int" } EQ_Contact(in1 := "Data_block_1".counter_datasuhu, in2 := 62)
      Move(in := "Suhu_Kanan", out1 => "Data_block_1".data_baru1[61])
   END_RUNG
   RUNG wire#w1
      { S7_Templates := "SrcType := Int" } EQ_Contact(in1 := "Data_block_1".counter_datasuhu, in2 := 63)
      Move(in := "Suhu_Kanan", out1 => "Data_block_1".data_baru1[62])
   END_RUNG
   RUNG wire#w1
      { S7_Templates := "SrcType := Int" } EQ_Contact(in1 := "Data_block_1".counter_datasuhu, in2 := 64)
      Move(in := "Suhu_Kanan", out1 => "Data_block_1".data_baru1[63])
   END_RUNG
   RUNG wire#w1
      { S7_Templates := "SrcType := Int" } EQ_Contact(in1 := "Data_block_1".counter_datasuhu, in2 := 65)
      Move(in := "Suhu_Kanan", out1 => "Data_block_1".data_baru1[64])
   END_RUNG
   RUNG wire#w1
      { S7_Templates := "SrcType := Int" } EQ_Contact(in1 := "Data_block_1".counter_datasuhu, in2 := 66)
      Move(in := "Suhu_Kanan", out1 => "Data_block_1".data_baru1[65])
   END_RUNG
   RUNG wire#w1
      { S7_Templates := "SrcType := Int" } EQ_Contact(in1 := "Data_block_1".counter_datasuhu, in2 := 67)
      Move(in := "Suhu_Kanan", out1 => "Data_block_1".data_baru1[66])
   END_RUNG
   RUNG wire#w1
      { S7_Templates := "SrcType := Int" } EQ_Contact(in1 := "Data_block_1".counter_datasuhu, in2 := 68)
      Move(in := "Suhu_Kanan", out1 => "Data_block_1".data_baru1[67])
   END_RUNG
   RUNG wire#w1
      { S7_Templates := "SrcType := Int" } EQ_Contact(in1 := "Data_block_1".counter_datasuhu, in2 := 69)
      Move(in := "Suhu_Kanan", out1 => "Data_block_1".data_baru1[68])
   END_RUNG
   RUNG wire#w1
      { S7_Templates := "SrcType := Int" } EQ_Contact(in1 := "Data_block_1".counter_datasuhu, in2 := 70)
      Move(in := "Suhu_Kanan", out1 => "Data_block_1".data_baru1[69])
   END_RUNG
   RUNG wire#w1
      { S7_Templates := "SrcType := Int" } EQ_Contact(in1 := "Data_block_1".counter_datasuhu, in2 := 71)
      Move(in := "Suhu_Kanan", out1 => "Data_block_1".data_baru1[70])
   END_RUNG
   RUNG wire#w1
      { S7_Templates := "SrcType := Int" } EQ_Contact(in1 := "Data_block_1".counter_datasuhu, in2 := 72)
      Move(in := "Suhu_Kanan", out1 => "Data_block_1".data_baru1[71])
   END_RUNG
   RUNG wire#w1
      { S7_Templates := "SrcType := Int" } EQ_Contact(in1 := "Data_block_1".counter_datasuhu, in2 := 73)
      Move(in := "Suhu_Kanan", out1 => "Data_block_1".data_baru1[72])
   END_RUNG
   RUNG wire#w1
      { S7_Templates := "SrcType := Int" } EQ_Contact(in1 := "Data_block_1".counter_datasuhu, in2 := 74)
      Move(in := "Suhu_Kanan", out1 => "Data_block_1".data_baru1[73])
   END_RUNG
   RUNG wire#w1
      { S7_Templates := "SrcType := Int" } EQ_Contact(in1 := "Data_block_1".counter_datasuhu, in2 := 75)
      Move(in := "Suhu_Kanan", out1 => "Data_block_1".data_baru1[74])
   END_RUNG
   RUNG wire#w1
      { S7_Templates := "SrcType := Int" } EQ_Contact(in1 := "Data_block_1".counter_datasuhu, in2 := 76)
      Move(in := "Suhu_Kanan", out1 => "Data_block_1".data_baru1[75])
   END_RUNG
   RUNG wire#w1
      { S7_Templates := "SrcType := Int" } EQ_Contact(in1 := "Data_block_1".counter_datasuhu, in2 := 77)
      Move(in := "Suhu_Kanan", out1 => "Data_block_1".data_baru1[76])
   END_RUNG
   RUNG wire#w1
      { S7_Templates := "SrcType := Int" } EQ_Contact(in1 := "Data_block_1".counter_datasuhu, in2 := 78)
      Move(in := "Suhu_Kanan", out1 => "Data_block_1".data_baru1[77])
   END_RUNG
   RUNG wire#w1
      { S7_Templates := "SrcType := Int" } EQ_Contact(in1 := "Data_block_1".counter_datasuhu, in2 := 79)
      Move(in := "Suhu_Kanan", out1 => "Data_block_1".data_baru1[78])
   END_RUNG
   RUNG wire#w1
      { S7_Templates := "SrcType := Int" } EQ_Contact(in1 := "Data_block_1".counter_datasuhu, in2 := 80)
      Move(in := "Suhu_Kanan", out1 => "Data_block_1".data_baru1[81])
   END_RUNG
   RUNG wire#w1
      { S7_Templates := "SrcType := Int" } EQ_Contact(in1 := "Data_block_1".counter_datasuhu, in2 := 81)
      Move(in := "Suhu_Kanan", out1 => "Data_block_1".data_baru1[80])
   END_RUNG
   RUNG wire#w1
      { S7_Templates := "SrcType := Int" } EQ_Contact(in1 := "Data_block_1".counter_datasuhu, in2 := 82)
      Move(in := "Suhu_Kanan", out1 => "Data_block_1".data_baru1[81])
   END_RUNG
   RUNG wire#w1
      { S7_Templates := "SrcType := Int" } EQ_Contact(in1 := "Data_block_1".counter_datasuhu, in2 := 83)
      Move(in := "Suhu_Kanan", out1 => "Data_block_1".data_baru1[82])
   END_RUNG
   RUNG wire#w1
      { S7_Templates := "SrcType := Int" } EQ_Contact(in1 := "Data_block_1".counter_datasuhu, in2 := 84)
      Move(in := "Suhu_Kanan", out1 => "Data_block_1".data_baru1[83])
   END_RUNG
   RUNG wire#w1
      { S7_Templates := "SrcType := Int" } EQ_Contact(in1 := "Data_block_1".counter_datasuhu, in2 := 85)
      Move(in := "Suhu_Kanan", out1 => "Data_block_1".data_baru1[84])
   END_RUNG
   RUNG wire#w1
      { S7_Templates := "SrcType := Int" } EQ_Contact(in1 := "Data_block_1".counter_datasuhu, in2 := 86)
      Move(in := "Suhu_Kanan", out1 => "Data_block_1".data_baru1[85])
   END_RUNG
   RUNG wire#w1
      { S7_Templates := "SrcType := Int" } EQ_Contact(in1 := "Data_block_1".counter_datasuhu, in2 := 87)
      Move(in := "Suhu_Kanan", out1 => "Data_block_1".data_baru1[86])
   END_RUNG
   RUNG wire#w1
      { S7_Templates := "SrcType := Int" } EQ_Contact(in1 := "Data_block_1".counter_datasuhu, in2 := 88)
      Move(in := "Suhu_Kanan", out1 => "Data_block_1".data_baru1[87])
   END_RUNG
   RUNG wire#w1
      { S7_Templates := "SrcType := Int" } EQ_Contact(in1 := "Data_block_1".counter_datasuhu, in2 := 89)
      Move(in := "Suhu_Kanan", out1 => "Data_block_1".data_baru1[88])
   END_RUNG
   RUNG wire#w1
      { S7_Templates := "SrcType := Int" } EQ_Contact(in1 := "Data_block_1".counter_datasuhu, in2 := 90)
      Move(in := "Suhu_Kanan", out1 => "Data_block_1".data_baru1[89])
   END_RUNG
   RUNG wire#w1
      { S7_Templates := "SrcType := Int" } EQ_Contact(in1 := "Data_block_1".counter_datasuhu, in2 := 91)
      Move(in := "Suhu_Kanan", out1 => "Data_block_1".data_baru1[90])
   END_RUNG
   RUNG wire#w1
      { S7_Templates := "SrcType := Int" } EQ_Contact(in1 := "Data_block_1".counter_datasuhu, in2 := 92)
      Move(in := "Suhu_Kanan", out1 => "Data_block_1".data_baru1[91])
   END_RUNG
   RUNG wire#w1
      { S7_Templates := "SrcType := Int" } EQ_Contact(in1 := "Data_block_1".counter_datasuhu, in2 := 93)
      Move(in := "Suhu_Kanan", out1 => "Data_block_1".data_baru1[92])
   END_RUNG
   RUNG wire#w1
      { S7_Templates := "SrcType := Int" } EQ_Contact(in1 := "Data_block_1".counter_datasuhu, in2 := 94)
      Move(in := "Suhu_Kanan", out1 => "Data_block_1".data_baru1[93])
   END_RUNG
   RUNG wire#w1
      { S7_Templates := "SrcType := Int" } EQ_Contact(in1 := "Data_block_1".counter_datasuhu, in2 := 95)
      Move(in := "Suhu_Kanan", out1 => "Data_block_1".data_baru1[94])
   END_RUNG
   RUNG wire#w1
      { S7_Templates := "SrcType := Int" } EQ_Contact(in1 := "Data_block_1".counter_datasuhu, in2 := 96)
      Move(in := "Suhu_Kanan", out1 => "Data_block_1".data_baru1[95])
   END_RUNG
   RUNG wire#w1
      { S7_Templates := "SrcType := Int" } EQ_Contact(in1 := "Data_block_1".counter_datasuhu, in2 := 97)
      Move(in := "Suhu_Kanan", out1 => "Data_block_1".data_baru1[96])
   END_RUNG
   RUNG wire#w1
      { S7_Templates := "SrcType := Int" } EQ_Contact(in1 := "Data_block_1".counter_datasuhu, in2 := 98)
      Move(in := "Suhu_Kanan", out1 => "Data_block_1".data_baru1[97])
   END_RUNG
   RUNG wire#w1
      { S7_Templates := "SrcType := Int" } EQ_Contact(in1 := "Data_block_1".counter_datasuhu, in2 := 99)
      Move(in := "Suhu_Kanan", out1 => "Data_block_1".data_baru1[98])
   END_RUNG
   RUNG wire#w1
      { S7_Templates := "SrcType := Int" } EQ_Contact(in1 := "Data_block_1".counter_datasuhu, in2 := 100)
      Move(in := "Suhu_Kanan", out1 => "Data_block_1".data_baru1[99])
   END_RUNG
   // the same network as SCL:
   #_w1 := "Data_block_1".K1 AND NOT "Data_block_1".Lock_B;
   IF #_w1 AND ("Data_block_1".counter_datasuhu = 1) THEN
       "Data_block_1".data_baru1[0] := "Suhu_Kanan";
   END_IF;
   IF #_w1 AND ("Data_block_1".counter_datasuhu = 2) THEN
       "Data_block_1".data_baru1[1] := "Suhu_Kanan";
   END_IF;
   IF #_w1 AND ("Data_block_1".counter_datasuhu = 3) THEN
       "Data_block_1".data_baru1[2] := "Suhu_Kanan";
   END_IF;
   IF #_w1 AND ("Data_block_1".counter_datasuhu = 4) THEN
       "Data_block_1".data_baru1[3] := "Suhu_Kanan";
   END_IF;
   IF #_w1 AND ("Data_block_1".counter_datasuhu = 5) THEN
       "Data_block_1".data_baru1[4] := "Suhu_Kanan";
   END_IF;
   IF #_w1 AND ("Data_block_1".counter_datasuhu = 6) THEN
       "Data_block_1".data_baru1[5] := "Suhu_Kanan";
   END_IF;
   IF #_w1 AND ("Data_block_1".counter_datasuhu = 7) THEN
       "Data_block_1".data_baru1[6] := "Suhu_Kanan";
   END_IF;
   IF #_w1 AND ("Data_block_1".counter_datasuhu = 8) THEN
       "Data_block_1".data_baru1[7] := "Suhu_Kanan";
   END_IF;
   IF #_w1 AND ("Data_block_1".counter_datasuhu = 9) THEN
       "Data_block_1".data_baru1[8] := "Suhu_Kanan";
   END_IF;
   IF #_w1 AND ("Data_block_1".counter_datasuhu = 10) THEN
       "Data_block_1".data_baru1[9] := "Suhu_Kanan";
   END_IF;
   IF #_w1 AND ("Data_block_1".counter_datasuhu = 11) THEN
       "Data_block_1".data_baru1[10] := "Suhu_Kanan";
   END_IF;
   IF #_w1 AND ("Data_block_1".counter_datasuhu = 12) THEN
       "Data_block_1".data_baru1[11] := "Suhu_Kanan";
   END_IF;
   IF #_w1 AND ("Data_block_1".counter_datasuhu = 13) THEN
       "Data_block_1".data_baru1[12] := "Suhu_Kanan";
   END_IF;
   IF #_w1 AND ("Data_block_1".counter_datasuhu = 14) THEN
       "Data_block_1".data_baru1[13] := "Suhu_Kanan";
   END_IF;
   IF #_w1 AND ("Data_block_1".counter_datasuhu = 15) THEN
       "Data_block_1".data_baru1[14] := "Suhu_Kanan";
   END_IF;
   IF #_w1 AND ("Data_block_1".counter_datasuhu = 16) THEN
       "Data_block_1".data_baru1[15] := "Suhu_Kanan";
   END_IF;
   IF #_w1 AND ("Data_block_1".counter_datasuhu = 17) THEN
       "Data_block_1".data_baru1[16] := "Suhu_Kanan";
   END_IF;
   IF #_w1 AND ("Data_block_1".counter_datasuhu = 18) THEN
       "Data_block_1".data_baru1[17] := "Suhu_Kanan";
   END_IF;
   IF #_w1 AND ("Data_block_1".counter_datasuhu = 19) THEN
       "Data_block_1".data_baru1[18] := "Suhu_Kanan";
   END_IF;
   IF #_w1 AND ("Data_block_1".counter_datasuhu = 20) THEN
       "Data_block_1".data_baru1[19] := "Suhu_Kanan";
   END_IF;
   IF #_w1 AND ("Data_block_1".counter_datasuhu = 21) THEN
       "Data_block_1".data_baru1[20] := "Suhu_Kanan";
   END_IF;
   IF #_w1 AND ("Data_block_1".counter_datasuhu = 22) THEN
       "Data_block_1".data_baru1[21] := "Suhu_Kanan";
   END_IF;
   IF #_w1 AND ("Data_block_1".counter_datasuhu = 23) THEN
       "Data_block_1".data_baru1[22] := "Suhu_Kanan";
   END_IF;
   IF #_w1 AND ("Data_block_1".counter_datasuhu = 24) THEN
       "Data_block_1".data_baru1[23] := "Suhu_Kanan";
   END_IF;
   IF #_w1 AND ("Data_block_1".counter_datasuhu = 25) THEN
       "Data_block_1".data_baru1[24] := "Suhu_Kanan";
   END_IF;
   IF #_w1 AND ("Data_block_1".counter_datasuhu = 26) THEN
       "Data_block_1".data_baru1[25] := "Suhu_Kanan";
   END_IF;
   IF #_w1 AND ("Data_block_1".counter_datasuhu = 27) THEN
       "Data_block_1".data_baru1[26] := "Suhu_Kanan";
   END_IF;
   IF #_w1 AND ("Data_block_1".counter_datasuhu = 28) THEN
       "Data_block_1".data_baru1[27] := "Suhu_Kanan";
   END_IF;
   IF #_w1 AND ("Data_block_1".counter_datasuhu = 29) THEN
       "Data_block_1".data_baru1[28] := "Suhu_Kanan";
   END_IF;
   IF #_w1 AND ("Data_block_1".counter_datasuhu = 30) THEN
       "Data_block_1".data_baru1[29] := "Suhu_Kanan";
   END_IF;
   IF #_w1 AND ("Data_block_1".counter_datasuhu = 31) THEN
       "Data_block_1".data_baru1[30] := "Suhu_Kanan";
   END_IF;
   IF #_w1 AND ("Data_block_1".counter_datasuhu = 32) THEN
       "Data_block_1".data_baru1[31] := "Suhu_Kanan";
   END_IF;
   IF #_w1 AND ("Data_block_1".counter_datasuhu = 33) THEN
       "Data_block_1".data_baru1[32] := "Suhu_Kanan";
   END_IF;
   IF #_w1 AND ("Data_block_1".counter_datasuhu = 34) THEN
       "Data_block_1".data_baru1[33] := "Suhu_Kanan";
   END_IF;
   IF #_w1 AND ("Data_block_1".counter_datasuhu = 35) THEN
       "Data_block_1".data_baru1[34] := "Suhu_Kanan";
   END_IF;
   IF #_w1 AND ("Data_block_1".counter_datasuhu = 36) THEN
       "Data_block_1".data_baru1[35] := "Suhu_Kanan";
   END_IF;
   IF #_w1 AND ("Data_block_1".counter_datasuhu = 37) THEN
       "Data_block_1".data_baru1[36] := "Suhu_Kanan";
   END_IF;
   IF #_w1 AND ("Data_block_1".counter_datasuhu = 38) THEN
       "Data_block_1".data_baru1[37] := "Suhu_Kanan";
   END_IF;
   IF #_w1 AND ("Data_block_1".counter_datasuhu = 39) THEN
       "Data_block_1".data_baru1[38] := "Suhu_Kanan";
   END_IF;
   IF #_w1 AND ("Data_block_1".counter_datasuhu = 40) THEN
       "Data_block_1".data_baru1[39] := "Suhu_Kanan";
   END_IF;
   IF #_w1 AND ("Data_block_1".counter_datasuhu = 41) THEN
       "Data_block_1".data_baru1[40] := "Suhu_Kanan";
   END_IF;
   IF #_w1 AND ("Data_block_1".counter_datasuhu = 42) THEN
       "Data_block_1".data_baru1[41] := "Suhu_Kanan";
   END_IF;
   IF #_w1 AND ("Data_block_1".counter_datasuhu = 43) THEN
       "Data_block_1".data_baru1[42] := "Suhu_Kanan";
   END_IF;
   IF #_w1 AND ("Data_block_1".counter_datasuhu = 44) THEN
       "Data_block_1".data_baru1[43] := "Suhu_Kanan";
   END_IF;
   IF #_w1 AND ("Data_block_1".counter_datasuhu = 45) THEN
       "Data_block_1".data_baru1[44] := "Suhu_Kanan";
   END_IF;
   IF #_w1 AND ("Data_block_1".counter_datasuhu = 46) THEN
       "Data_block_1".data_baru1[45] := "Suhu_Kanan";
   END_IF;
   IF #_w1 AND ("Data_block_1".counter_datasuhu = 47) THEN
       "Data_block_1".data_baru1[46] := "Suhu_Kanan";
   END_IF;
   IF #_w1 AND ("Data_block_1".counter_datasuhu = 48) THEN
       "Data_block_1".data_baru1[47] := "Suhu_Kanan";
   END_IF;
   IF #_w1 AND ("Data_block_1".counter_datasuhu = 49) THEN
       "Data_block_1".data_baru1[48] := "Suhu_Kanan";
   END_IF;
   IF #_w1 AND ("Data_block_1".counter_datasuhu = 50) THEN
       "Data_block_1".data_baru1[49] := "Suhu_Kanan";
   END_IF;
   IF #_w1 AND ("Data_block_1".counter_datasuhu = 51) THEN
       "Data_block_1".data_baru1[50] := "Suhu_Kanan";
   END_IF;
   IF #_w1 AND ("Data_block_1".counter_datasuhu = 52) THEN
       "Data_block_1".data_baru1[51] := "Suhu_Kanan";
   END_IF;
   IF #_w1 AND ("Data_block_1".counter_datasuhu = 53) THEN
       "Data_block_1".data_baru1[52] := "Suhu_Kanan";
   END_IF;
   IF #_w1 AND ("Data_block_1".counter_datasuhu = 54) THEN
       "Data_block_1".data_baru1[53] := "Suhu_Kanan";
   END_IF;
   IF #_w1 AND ("Data_block_1".counter_datasuhu = 55) THEN
       "Data_block_1".data_baru1[54] := "Suhu_Kanan";
   END_IF;
   IF #_w1 AND ("Data_block_1".counter_datasuhu = 56) THEN
       "Data_block_1".data_baru1[55] := "Suhu_Kanan";
   END_IF;
   IF #_w1 AND ("Data_block_1".counter_datasuhu = 57) THEN
       "Data_block_1".data_baru1[56] := "Suhu_Kanan";
   END_IF;
   IF #_w1 AND ("Data_block_1".counter_datasuhu = 58) THEN
       "Data_block_1".data_baru1[57] := "Suhu_Kanan";
   END_IF;
   IF #_w1 AND ("Data_block_1".counter_datasuhu = 59) THEN
       "Data_block_1".data_baru1[58] := "Suhu_Kanan";
   END_IF;
   IF #_w1 AND ("Data_block_1".counter_datasuhu = 60) THEN
       "Data_block_1".data_baru1[59] := "Suhu_Kanan";
   END_IF;
   IF #_w1 AND ("Data_block_1".counter_datasuhu = 61) THEN
       "Data_block_1".data_baru1[60] := "Suhu_Kanan";
   END_IF;
   IF #_w1 AND ("Data_block_1".counter_datasuhu = 62) THEN
       "Data_block_1".data_baru1[61] := "Suhu_Kanan";
   END_IF;
   IF #_w1 AND ("Data_block_1".counter_datasuhu = 63) THEN
       "Data_block_1".data_baru1[62] := "Suhu_Kanan";
   END_IF;
   IF #_w1 AND ("Data_block_1".counter_datasuhu = 64) THEN
       "Data_block_1".data_baru1[63] := "Suhu_Kanan";
   END_IF;
   IF #_w1 AND ("Data_block_1".counter_datasuhu = 65) THEN
       "Data_block_1".data_baru1[64] := "Suhu_Kanan";
   END_IF;
   IF #_w1 AND ("Data_block_1".counter_datasuhu = 66) THEN
       "Data_block_1".data_baru1[65] := "Suhu_Kanan";
   END_IF;
   IF #_w1 AND ("Data_block_1".counter_datasuhu = 67) THEN
       "Data_block_1".data_baru1[66] := "Suhu_Kanan";
   END_IF;
   IF #_w1 AND ("Data_block_1".counter_datasuhu = 68) THEN
       "Data_block_1".data_baru1[67] := "Suhu_Kanan";
   END_IF;
   IF #_w1 AND ("Data_block_1".counter_datasuhu = 69) THEN
       "Data_block_1".data_baru1[68] := "Suhu_Kanan";
   END_IF;
   IF #_w1 AND ("Data_block_1".counter_datasuhu = 70) THEN
       "Data_block_1".data_baru1[69] := "Suhu_Kanan";
   END_IF;
   IF #_w1 AND ("Data_block_1".counter_datasuhu = 71) THEN
       "Data_block_1".data_baru1[70] := "Suhu_Kanan";
   END_IF;
   IF #_w1 AND ("Data_block_1".counter_datasuhu = 72) THEN
       "Data_block_1".data_baru1[71] := "Suhu_Kanan";
   END_IF;
   IF #_w1 AND ("Data_block_1".counter_datasuhu = 73) THEN
       "Data_block_1".data_baru1[72] := "Suhu_Kanan";
   END_IF;
   IF #_w1 AND ("Data_block_1".counter_datasuhu = 74) THEN
       "Data_block_1".data_baru1[73] := "Suhu_Kanan";
   END_IF;
   IF #_w1 AND ("Data_block_1".counter_datasuhu = 75) THEN
       "Data_block_1".data_baru1[74] := "Suhu_Kanan";
   END_IF;
   IF #_w1 AND ("Data_block_1".counter_datasuhu = 76) THEN
       "Data_block_1".data_baru1[75] := "Suhu_Kanan";
   END_IF;
   IF #_w1 AND ("Data_block_1".counter_datasuhu = 77) THEN
       "Data_block_1".data_baru1[76] := "Suhu_Kanan";
   END_IF;
   IF #_w1 AND ("Data_block_1".counter_datasuhu = 78) THEN
       "Data_block_1".data_baru1[77] := "Suhu_Kanan";
   END_IF;
   IF #_w1 AND ("Data_block_1".counter_datasuhu = 79) THEN
       "Data_block_1".data_baru1[78] := "Suhu_Kanan";
   END_IF;
   IF #_w1 AND ("Data_block_1".counter_datasuhu = 80) THEN
       "Data_block_1".data_baru1[81] := "Suhu_Kanan";
   END_IF;
   IF #_w1 AND ("Data_block_1".counter_datasuhu = 81) THEN
       "Data_block_1".data_baru1[80] := "Suhu_Kanan";
   END_IF;
   IF #_w1 AND ("Data_block_1".counter_datasuhu = 82) THEN
       "Data_block_1".data_baru1[81] := "Suhu_Kanan";
   END_IF;
   IF #_w1 AND ("Data_block_1".counter_datasuhu = 83) THEN
       "Data_block_1".data_baru1[82] := "Suhu_Kanan";
   END_IF;
   IF #_w1 AND ("Data_block_1".counter_datasuhu = 84) THEN
       "Data_block_1".data_baru1[83] := "Suhu_Kanan";
   END_IF;
   IF #_w1 AND ("Data_block_1".counter_datasuhu = 85) THEN
       "Data_block_1".data_baru1[84] := "Suhu_Kanan";
   END_IF;
   IF #_w1 AND ("Data_block_1".counter_datasuhu = 86) THEN
       "Data_block_1".data_baru1[85] := "Suhu_Kanan";
   END_IF;
   IF #_w1 AND ("Data_block_1".counter_datasuhu = 87) THEN
       "Data_block_1".data_baru1[86] := "Suhu_Kanan";
   END_IF;
   IF #_w1 AND ("Data_block_1".counter_datasuhu = 88) THEN
       "Data_block_1".data_baru1[87] := "Suhu_Kanan";
   END_IF;
   IF #_w1 AND ("Data_block_1".counter_datasuhu = 89) THEN
       "Data_block_1".data_baru1[88] := "Suhu_Kanan";
   END_IF;
   IF #_w1 AND ("Data_block_1".counter_datasuhu = 90) THEN
       "Data_block_1".data_baru1[89] := "Suhu_Kanan";
   END_IF;
   IF #_w1 AND ("Data_block_1".counter_datasuhu = 91) THEN
       "Data_block_1".data_baru1[90] := "Suhu_Kanan";
   END_IF;
   IF #_w1 AND ("Data_block_1".counter_datasuhu = 92) THEN
       "Data_block_1".data_baru1[91] := "Suhu_Kanan";
   END_IF;
   IF #_w1 AND ("Data_block_1".counter_datasuhu = 93) THEN
       "Data_block_1".data_baru1[92] := "Suhu_Kanan";
   END_IF;
   IF #_w1 AND ("Data_block_1".counter_datasuhu = 94) THEN
       "Data_block_1".data_baru1[93] := "Suhu_Kanan";
   END_IF;
   IF #_w1 AND ("Data_block_1".counter_datasuhu = 95) THEN
       "Data_block_1".data_baru1[94] := "Suhu_Kanan";
   END_IF;
   IF #_w1 AND ("Data_block_1".counter_datasuhu = 96) THEN
       "Data_block_1".data_baru1[95] := "Suhu_Kanan";
   END_IF;
   IF #_w1 AND ("Data_block_1".counter_datasuhu = 97) THEN
       "Data_block_1".data_baru1[96] := "Suhu_Kanan";
   END_IF;
   IF #_w1 AND ("Data_block_1".counter_datasuhu = 98) THEN
       "Data_block_1".data_baru1[97] := "Suhu_Kanan";
   END_IF;
   IF #_w1 AND ("Data_block_1".counter_datasuhu = 99) THEN
       "Data_block_1".data_baru1[98] := "Suhu_Kanan";
   END_IF;
   IF #_w1 AND ("Data_block_1".counter_datasuhu = 100) THEN
       "Data_block_1".data_baru1[99] := "Suhu_Kanan";
   END_IF;
END_REGION

REGION Network 9: Data Pengambilan Suhu Per Roda
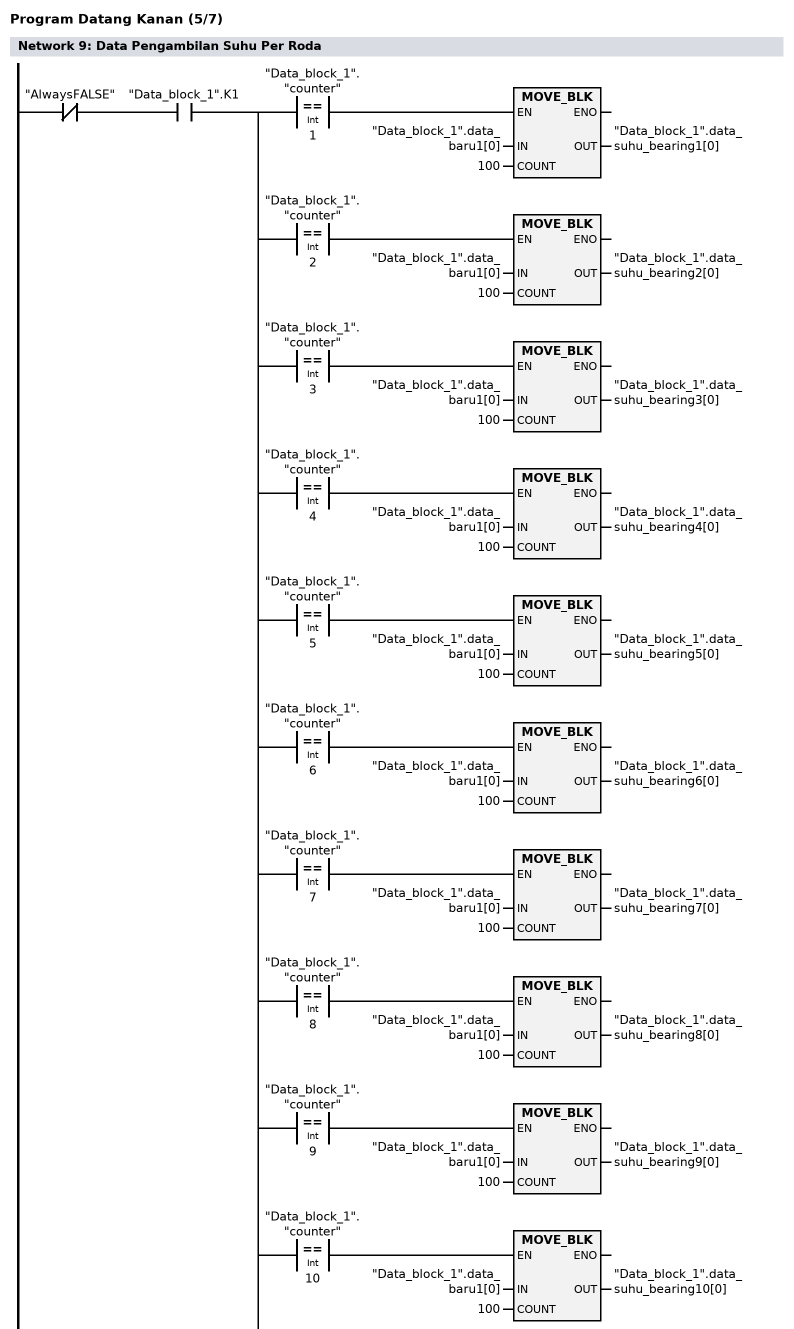
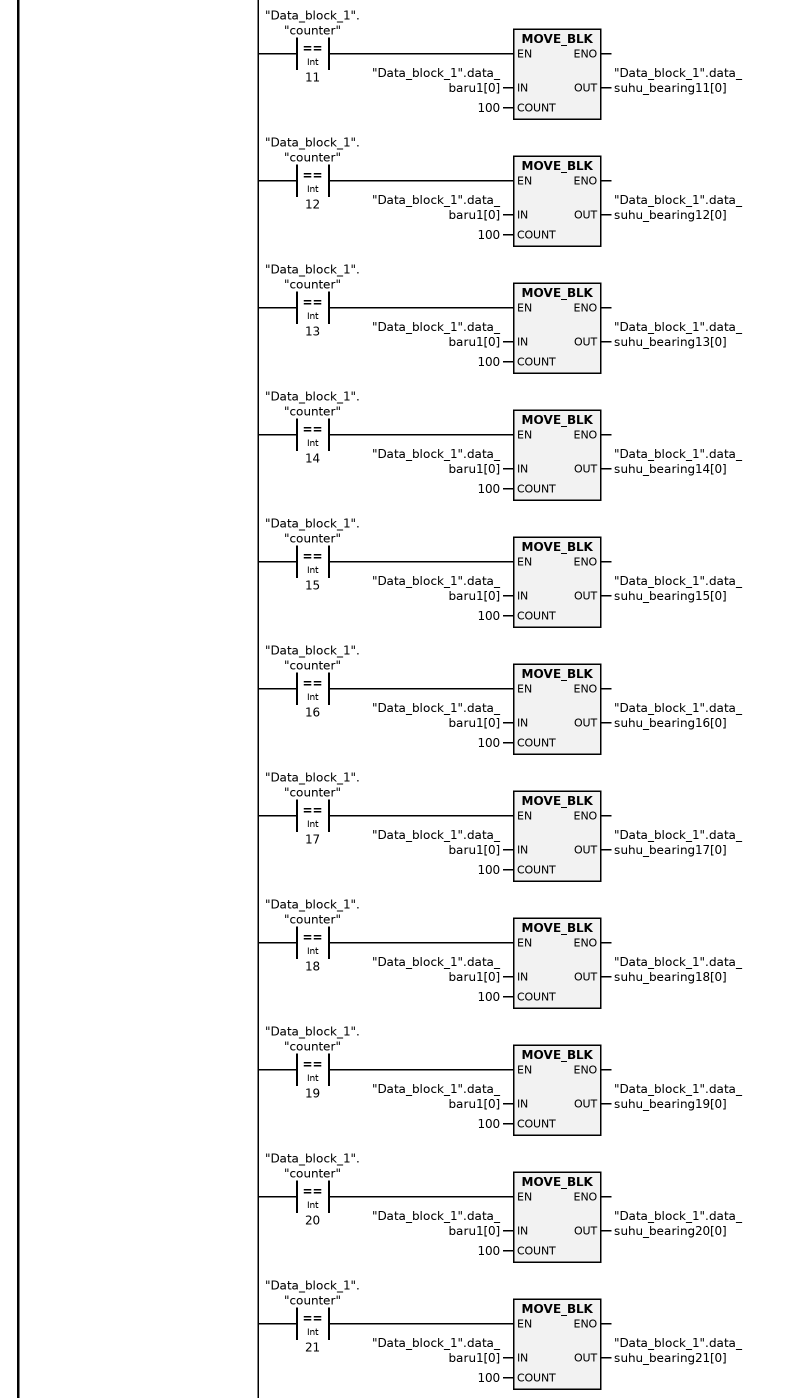
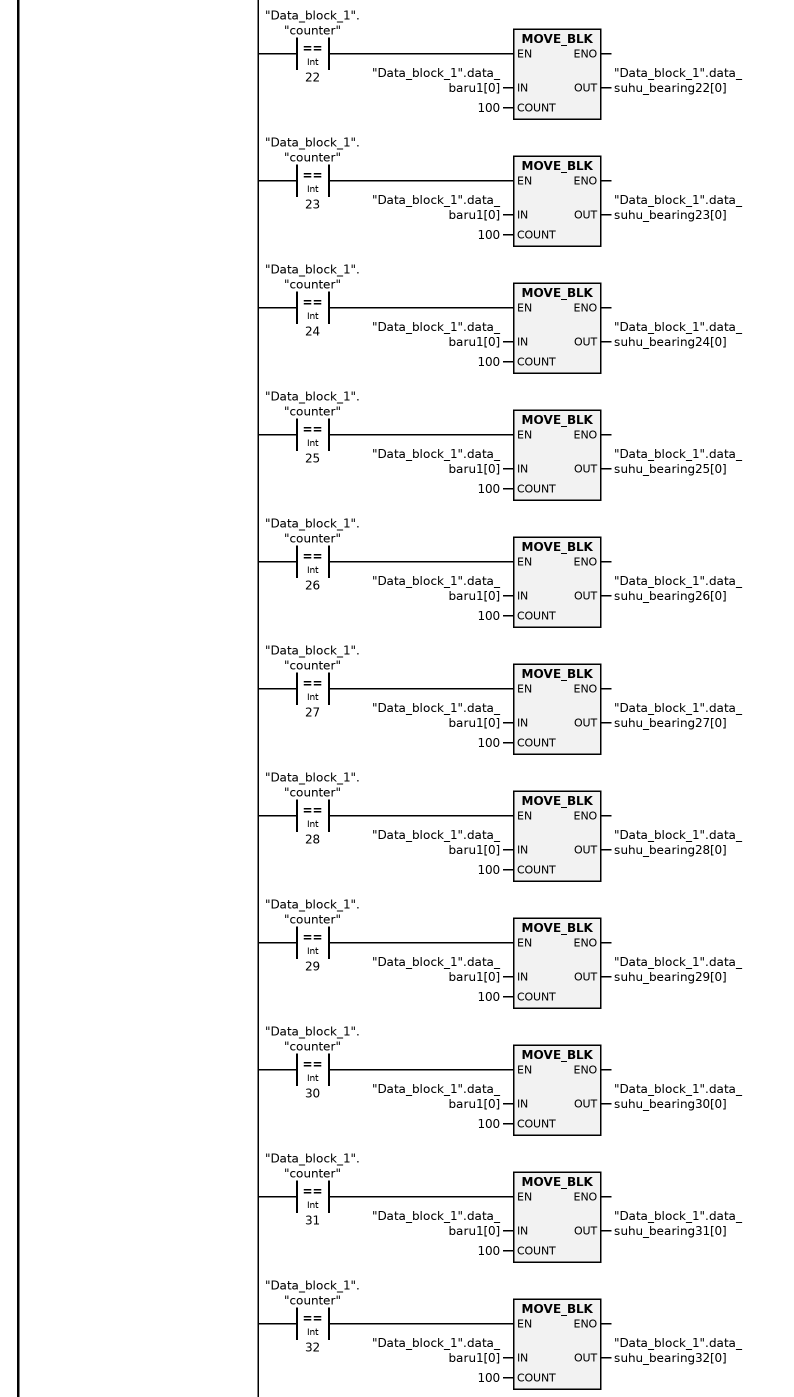
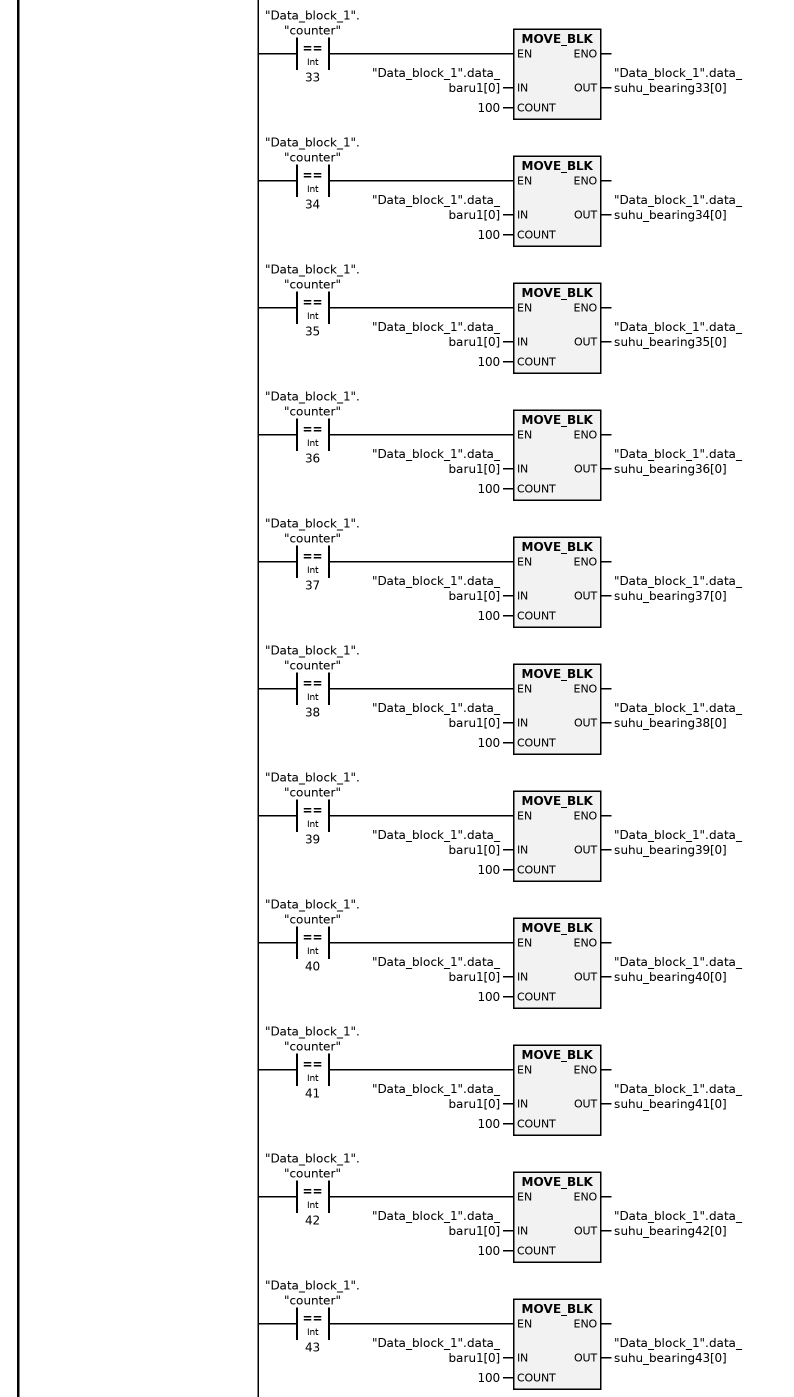
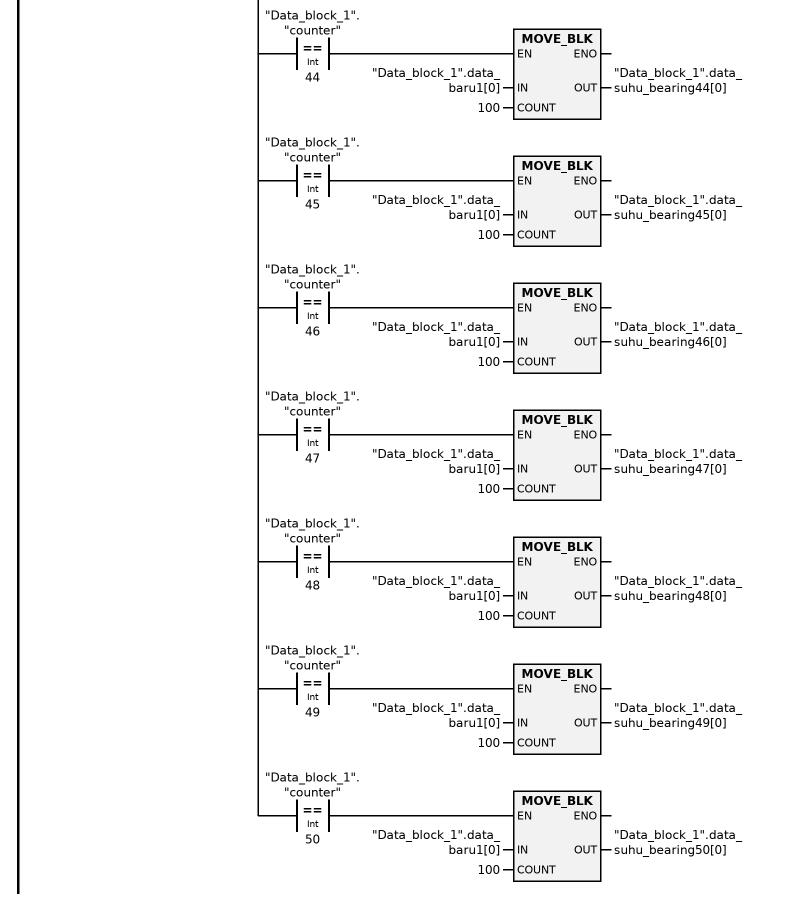
   #_w1 := NOT "AlwaysFALSE" AND "Data_block_1".K1;
   IF #_w1 AND ("Data_block_1"."counter" = 1) THEN
       MOVE_BLK(IN := "Data_block_1".data_baru1[0], COUNT := 100, OUT => "Data_block_1".data_suhu_bearing1[0]);
   END_IF;
   IF #_w1 AND ("Data_block_1"."counter" = 2) THEN
       MOVE_BLK(IN := "Data_block_1".data_baru1[0], COUNT := 100, OUT => "Data_block_1".data_suhu_bearing2[0]);
   END_IF;
   IF #_w1 AND ("Data_block_1"."counter" = 3) THEN
       MOVE_BLK(IN := "Data_block_1".data_baru1[0], COUNT := 100, OUT => "Data_block_1".data_suhu_bearing3[0]);
   END_IF;
   IF #_w1 AND ("Data_block_1"."counter" = 4) THEN
       MOVE_BLK(IN := "Data_block_1".data_baru1[0], COUNT := 100, OUT => "Data_block_1".data_suhu_bearing4[0]);
   END_IF;
   IF #_w1 AND ("Data_block_1"."counter" = 5) THEN
       MOVE_BLK(IN := "Data_block_1".data_baru1[0], COUNT := 100, OUT => "Data_block_1".data_suhu_bearing5[0]);
   END_IF;
   IF #_w1 AND ("Data_block_1"."counter" = 6) THEN
       MOVE_BLK(IN := "Data_block_1".data_baru1[0], COUNT := 100, OUT => "Data_block_1".data_suhu_bearing6[0]);
   END_IF;
   IF #_w1 AND ("Data_block_1"."counter" = 7) THEN
       MOVE_BLK(IN := "Data_block_1".data_baru1[0], COUNT := 100, OUT => "Data_block_1".data_suhu_bearing7[0]);
   END_IF;
   IF #_w1 AND ("Data_block_1"."counter" = 8) THEN
       MOVE_BLK(IN := "Data_block_1".data_baru1[0], COUNT := 100, OUT => "Data_block_1".data_suhu_bearing8[0]);
   END_IF;
   IF #_w1 AND ("Data_block_1"."counter" = 9) THEN
       MOVE_BLK(IN := "Data_block_1".data_baru1[0], COUNT := 100, OUT => "Data_block_1".data_suhu_bearing9[0]);
   END_IF;
   IF #_w1 AND ("Data_block_1"."counter" = 10) THEN
       MOVE_BLK(IN := "Data_block_1".data_baru1[0], COUNT := 100, OUT => "Data_block_1".data_suhu_bearing10[0]);
   END_IF;
   IF #_w1 AND ("Data_block_1"."counter" = 11) THEN
       MOVE_BLK(IN := "Data_block_1".data_baru1[0], COUNT := 100, OUT => "Data_block_1".data_suhu_bearing11[0]);
   END_IF;
   IF #_w1 AND ("Data_block_1"."counter" = 12) THEN
       MOVE_BLK(IN := "Data_block_1".data_baru1[0], COUNT := 100, OUT => "Data_block_1".data_suhu_bearing12[0]);
   END_IF;
   IF #_w1 AND ("Data_block_1"."counter" = 13) THEN
       MOVE_BLK(IN := "Data_block_1".data_baru1[0], COUNT := 100, OUT => "Data_block_1".data_suhu_bearing13[0]);
   END_IF;
   IF #_w1 AND ("Data_block_1"."counter" = 14) THEN
       MOVE_BLK(IN := "Data_block_1".data_baru1[0], COUNT := 100, OUT => "Data_block_1".data_suhu_bearing14[0]);
   END_IF;
   IF #_w1 AND ("Data_block_1"."counter" = 15) THEN
       MOVE_BLK(IN := "Data_block_1".data_baru1[0], COUNT := 100, OUT => "Data_block_1".data_suhu_bearing15[0]);
   END_IF;
   IF #_w1 AND ("Data_block_1"."counter" = 16) THEN
       MOVE_BLK(IN := "Data_block_1".data_baru1[0], COUNT := 100, OUT => "Data_block_1".data_suhu_bearing16[0]);
   END_IF;
   IF #_w1 AND ("Data_block_1"."counter" = 17) THEN
       MOVE_BLK(IN := "Data_block_1".data_baru1[0], COUNT := 100, OUT => "Data_block_1".data_suhu_bearing17[0]);
   END_IF;
   IF #_w1 AND ("Data_block_1"."counter" = 18) THEN
       MOVE_BLK(IN := "Data_block_1".data_baru1[0], COUNT := 100, OUT => "Data_block_1".data_suhu_bearing18[0]);
   END_IF;
   IF #_w1 AND ("Data_block_1"."counter" = 19) THEN
       MOVE_BLK(IN := "Data_block_1".data_baru1[0], COUNT := 100, OUT => "Data_block_1".data_suhu_bearing19[0]);
   END_IF;
   IF #_w1 AND ("Data_block_1"."counter" = 20) THEN
       MOVE_BLK(IN := "Data_block_1".data_baru1[0], COUNT := 100, OUT => "Data_block_1".data_suhu_bearing20[0]);
   END_IF;
   IF #_w1 AND ("Data_block_1"."counter" = 21) THEN
       MOVE_BLK(IN := "Data_block_1".data_baru1[0], COUNT := 100, OUT => "Data_block_1".data_suhu_bearing21[0]);
   END_IF;
   IF #_w1 AND ("Data_block_1"."counter" = 22) THEN
       MOVE_BLK(IN := "Data_block_1".data_baru1[0], COUNT := 100, OUT => "Data_block_1".data_suhu_bearing22[0]);
   END_IF;
   IF #_w1 AND ("Data_block_1"."counter" = 23) THEN
       MOVE_BLK(IN := "Data_block_1".data_baru1[0], COUNT := 100, OUT => "Data_block_1".data_suhu_bearing23[0]);
   END_IF;
   IF #_w1 AND ("Data_block_1"."counter" = 24) THEN
       MOVE_BLK(IN := "Data_block_1".data_baru1[0], COUNT := 100, OUT => "Data_block_1".data_suhu_bearing24[0]);
   END_IF;
   IF #_w1 AND ("Data_block_1"."counter" = 25) THEN
       MOVE_BLK(IN := "Data_block_1".data_baru1[0], COUNT := 100, OUT => "Data_block_1".data_suhu_bearing25[0]);
   END_IF;
   IF #_w1 AND ("Data_block_1"."counter" = 26) THEN
       MOVE_BLK(IN := "Data_block_1".data_baru1[0], COUNT := 100, OUT => "Data_block_1".data_suhu_bearing26[0]);
   END_IF;
   IF #_w1 AND ("Data_block_1"."counter" = 27) THEN
       MOVE_BLK(IN := "Data_block_1".data_baru1[0], COUNT := 100, OUT => "Data_block_1".data_suhu_bearing27[0]);
   END_IF;
   IF #_w1 AND ("Data_block_1"."counter" = 28) THEN
       MOVE_BLK(IN := "Data_block_1".data_baru1[0], COUNT := 100, OUT => "Data_block_1".data_suhu_bearing28[0]);
   END_IF;
   IF #_w1 AND ("Data_block_1"."counter" = 29) THEN
       MOVE_BLK(IN := "Data_block_1".data_baru1[0], COUNT := 100, OUT => "Data_block_1".data_suhu_bearing29[0]);
   END_IF;
   IF #_w1 AND ("Data_block_1"."counter" = 30) THEN
       MOVE_BLK(IN := "Data_block_1".data_baru1[0], COUNT := 100, OUT => "Data_block_1".data_suhu_bearing30[0]);
   END_IF;
   IF #_w1 AND ("Data_block_1"."counter" = 31) THEN
       MOVE_BLK(IN := "Data_block_1".data_baru1[0], COUNT := 100, OUT => "Data_block_1".data_suhu_bearing31[0]);
   END_IF;
   IF #_w1 AND ("Data_block_1"."counter" = 32) THEN
       MOVE_BLK(IN := "Data_block_1".data_baru1[0], COUNT := 100, OUT => "Data_block_1".data_suhu_bearing32[0]);
   END_IF;
   IF #_w1 AND ("Data_block_1"."counter" = 33) THEN
       MOVE_BLK(IN := "Data_block_1".data_baru1[0], COUNT := 100, OUT => "Data_block_1".data_suhu_bearing33[0]);
   END_IF;
   IF #_w1 AND ("Data_block_1"."counter" = 34) THEN
       MOVE_BLK(IN := "Data_block_1".data_baru1[0], COUNT := 100, OUT => "Data_block_1".data_suhu_bearing34[0]);
   END_IF;
   IF #_w1 AND ("Data_block_1"."counter" = 35) THEN
       MOVE_BLK(IN := "Data_block_1".data_baru1[0], COUNT := 100, OUT => "Data_block_1".data_suhu_bearing35[0]);
   END_IF;
   IF #_w1 AND ("Data_block_1"."counter" = 36) THEN
       MOVE_BLK(IN := "Data_block_1".data_baru1[0], COUNT := 100, OUT => "Data_block_1".data_suhu_bearing36[0]);
   END_IF;
   IF #_w1 AND ("Data_block_1"."counter" = 37) THEN
       MOVE_BLK(IN := "Data_block_1".data_baru1[0], COUNT := 100, OUT => "Data_block_1".data_suhu_bearing37[0]);
   END_IF;
   IF #_w1 AND ("Data_block_1"."counter" = 38) THEN
       MOVE_BLK(IN := "Data_block_1".data_baru1[0], COUNT := 100, OUT => "Data_block_1".data_suhu_bearing38[0]);
   END_IF;
   IF #_w1 AND ("Data_block_1"."counter" = 39) THEN
       MOVE_BLK(IN := "Data_block_1".data_baru1[0], COUNT := 100, OUT => "Data_block_1".data_suhu_bearing39[0]);
   END_IF;
   IF #_w1 AND ("Data_block_1"."counter" = 40) THEN
       MOVE_BLK(IN := "Data_block_1".data_baru1[0], COUNT := 100, OUT => "Data_block_1".data_suhu_bearing40[0]);
   END_IF;
   IF #_w1 AND ("Data_block_1"."counter" = 41) THEN
       MOVE_BLK(IN := "Data_block_1".data_baru1[0], COUNT := 100, OUT => "Data_block_1".data_suhu_bearing41[0]);
   END_IF;
   IF #_w1 AND ("Data_block_1"."counter" = 42) THEN
       MOVE_BLK(IN := "Data_block_1".data_baru1[0], COUNT := 100, OUT => "Data_block_1".data_suhu_bearing42[0]);
   END_IF;
   IF #_w1 AND ("Data_block_1"."counter" = 43) THEN
       MOVE_BLK(IN := "Data_block_1".data_baru1[0], COUNT := 100, OUT => "Data_block_1".data_suhu_bearing43[0]);
   END_IF;
   IF #_w1 AND ("Data_block_1"."counter" = 44) THEN
       MOVE_BLK(IN := "Data_block_1".data_baru1[0], COUNT := 100, OUT => "Data_block_1".data_suhu_bearing44[0]);
   END_IF;
   IF #_w1 AND ("Data_block_1"."counter" = 45) THEN
       MOVE_BLK(IN := "Data_block_1".data_baru1[0], COUNT := 100, OUT => "Data_block_1".data_suhu_bearing45[0]);
   END_IF;
   IF #_w1 AND ("Data_block_1"."counter" = 46) THEN
       MOVE_BLK(IN := "Data_block_1".data_baru1[0], COUNT := 100, OUT => "Data_block_1".data_suhu_bearing46[0]);
   END_IF;
   IF #_w1 AND ("Data_block_1"."counter" = 47) THEN
       MOVE_BLK(IN := "Data_block_1".data_baru1[0], COUNT := 100, OUT => "Data_block_1".data_suhu_bearing47[0]);
   END_IF;
   IF #_w1 AND ("Data_block_1"."counter" = 48) THEN
       MOVE_BLK(IN := "Data_block_1".data_baru1[0], COUNT := 100, OUT => "Data_block_1".data_suhu_bearing48[0]);
   END_IF;
   IF #_w1 AND ("Data_block_1"."counter" = 49) THEN
       MOVE_BLK(IN := "Data_block_1".data_baru1[0], COUNT := 100, OUT => "Data_block_1".data_suhu_bearing49[0]);
   END_IF;
   IF #_w1 AND ("Data_block_1"."counter" = 50) THEN
       MOVE_BLK(IN := "Data_block_1".data_baru1[0], COUNT := 100, OUT => "Data_block_1".data_suhu_bearing50[0]);
   END_IF;
END_REGION

REGION Network 10: Reset Data Suhu Per Roda
